KUKA KRL program: MyProgram_137().src

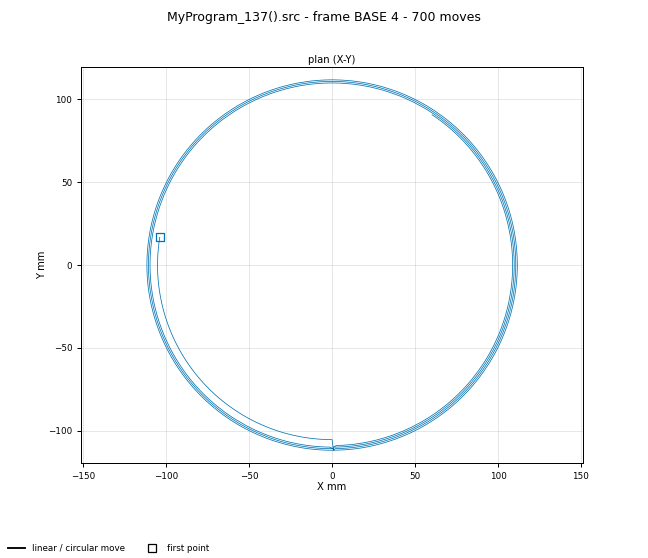
[picture p0: tool path of MyProgram_137().src in frame BASE 4, 700 of 700 moves have a stored position in this frame; points joined in program order, loops and branches not executed]
&ACCESS RVP
&REL 1
&PARAM TEMPLATE = C:\KRC\Roboter\Template\vorgabe
&PARAM EDITMASK = *
DEF MyProgram_137()
; ---- Setting reference (Base) ----
$BASE = BASE_DATA[4]

; --------------------------
; ---- Setting tool (TCP) ----
$TOOL = TOOL_DATA[3]
; --------------------------

$VEL.CP = VEL_APROX_PRINT
Startdeposition()
$VEL.CP = VEL_PRINT
LIN {X -103.9153,Y 16.7331,Z 110,A 166.763,B 24.9342,C -1.8738,E1 24.8417,E2 278.8329} C_DIS
LIN {X -104.4625,Y 12.8836,Z 110,A 168.8977,B 24.9346,C -1.8676,E1 24.8409,E2 276.7001} C_DIS
LIN {X -104.7464,Y 10.3245,Z 110,A 170.3073,B 24.9349,C -1.8633,E1 24.8405,E2 275.2923} C_DIS
LIN {X -104.9675,Y 7.7597,Z 110,A 171.7211,B 24.9352,C -1.8592,E1 24.8401,E2 273.8797} C_DIS
LIN {X -105.1015,Y 5.6308,Z 110,A 172.9515,B 24.9352,C -1.858,E1 24.84,E2 272.6448} C_DIS
LIN {X -105.2376,Y 1.7511,Z 110,A 174.9774,B 24.936,C -1.848,E1 24.8398,E2 270.6305} C_DIS
LIN {X -105.2498,Y -0.7552,Z 110,A 176.4837,B 24.936,C -1.8487,E1 24.8398,E2 269.1135} C_DIS
LIN {X -105.1831,Y -3.8616,Z 110,A 178.2625,B 24.936,C -1.8464,E1 24.84,E2 267.3295} C_DIS
LIN {X -105.0018,Y -7.2556,Z 110,A 179.9647,B 24.9369,C -1.8351,E1 24.8402,E2 265.6439} C_DIS
LIN {X -104.7784,Y -9.9782,Z 110,A -178.5617,B 24.9372,C -1.8299,E1 24.8406,E2 264.1741} C_DIS
LIN {X -104.4634,Y -12.8763,Z 110,A -176.7775,B 24.9371,C -1.8319,E1 24.8412,E2 262.3742} C_DIS
LIN {X -104.0207,Y -16.0526,Z 110,A -175.1402,B 24.9377,C -1.8225,E1 24.8419,E2 260.7497} C_DIS
LIN {X -103.4748,Y -19.271,Z 110,A -173.4007,B 24.9382,C -1.8155,E1 24.8427,E2 259.0165} C_DIS
LIN {X -102.6969,Y -23.0595,Z 110,A -171.2783,B 24.9386,C -1.8096,E1 24.8439,E2 256.8958} C_DIS
LIN {X -102.0023,Y -25.9537,Z 110,A -169.5758,B 24.9388,C -1.8076,E1 24.8451,E2 255.1881} C_DIS
LIN {X -101.2146,Y -28.8725,Z 110,A -167.9294,B 24.9391,C -1.8026,E1 24.8463,E2 253.5441} C_DIS
LIN {X -100.477,Y -31.3431,Z 110,A -166.5162,B 24.9394,C -1.7987,E1 24.8475,E2 252.132} C_DIS
LIN {X -99.3778,Y -34.6711,Z 110,A -164.5611,B 24.9396,C -1.7947,E1 24.8492,E2 250.1753} C_DIS
LIN {X -98.2809,Y -37.67,Z 110,A -162.7314,B 24.9398,C -1.7929,E1 24.851,E2 248.3396} C_DIS
LIN {X -96.9545,Y -40.9612,Z 110,A -160.9726,B 24.9405,C -1.781,E1 24.8529,E2 246.5994} C_DIS
LIN {X -95.6958,Y -43.8259,Z 110,A -159.2509,B 24.9408,C -1.7767,E1 24.8548,E2 244.8784} C_DIS
LIN {X -94.0154,Y -47.3234,Z 110,A -157.1242,B 24.9412,C -1.7713,E1 24.8574,E2 242.7531} C_DIS
LIN {X -92.2133,Y -50.7454,Z 110,A -155.0081,B 24.9416,C -1.7659,E1 24.8602,E2 240.6386} C_DIS
LIN {X -90.2743,Y -54.1198,Z 110,A -152.8768,B 24.9419,C -1.7607,E1 24.8632,E2 238.5087} C_DIS
LIN {X -88.4772,Y -57.0071,Z 110,A -150.9522,B 24.942,C -1.7586,E1 24.8661,E2 236.5793} C_DIS
LIN {X -86.4702,Y -60.0076,Z 110,A -148.9751,B 24.9423,C -1.754,E1 24.8692,E2 234.6033} C_DIS
LIN {X -84.5433,Y -62.6964,Z 110,A -147.1303,B 24.9425,C -1.7512,E1 24.8722,E2 232.7564} C_DIS
LIN {X -82.5713,Y -65.2685,Z 110,A -145.3762,B 24.9428,C -1.7466,E1 24.8752,E2 231.005} C_DIS
LIN {X -80.5409,Y -67.7611,Z 110,A -143.5381,B 24.9428,C -1.7457,E1 24.8785,E2 229.1605} C_DIS
LIN {X -78.4313,Y -70.1892,Z 110,A -141.8851,B 24.9434,C -1.7381,E1 24.8816,E2 227.5181} C_DIS
LIN {X -76.0517,Y -72.7618,Z 110,A -139.8973,B 24.9434,C -1.7369,E1 24.8854,E2 225.5246} C_DIS
LIN {X -73.6749,Y -75.1676,Z 110,A -137.9924,B 24.9436,C -1.7354,E1 24.8892,E2 223.6152} C_DIS
LIN {X -71.1541,Y -77.5569,Z 110,A -136.1922,B 24.944,C -1.7281,E1 24.8928,E2 221.8249} C_DIS
LIN {X -68.4428,Y -79.9602,Z 110,A -134.2214,B 24.9443,C -1.7242,E1 24.897,E2 219.8558} C_DIS
LIN {X -65.975,Y -82.0088,Z 110,A -132.4324,B 24.9443,C -1.7225,E1 24.9008,E2 218.0638} C_DIS
LIN {X -63.2601,Y -84.1199,Z 110,A -130.6012,B 24.9447,C -1.7177,E1 24.9049,E2 216.2377} C_DIS
LIN {X -60.6051,Y -86.0548,Z 110,A -128.8602,B 24.945,C -1.7128,E1 24.9088,E2 214.5022} C_DIS
LIN {X -58.8664,Y -87.2512,Z 110,A -127.6452,B 24.945,C -1.7135,E1 24.9116,E2 213.2815} C_DIS
LIN {X -55.9198,Y -89.1684,Z 110,A -125.7403,B 24.9452,C -1.7102,E1 24.9161,E2 211.3784} C_DIS
LIN {X -53.3923,Y -90.7044,Z 110,A -124.1717,B 24.9454,C -1.7062,E1 24.9199,E2 209.8144} C_DIS
LIN {X -50.7507,Y -92.2105,Z 110,A -122.5116,B 24.9456,C -1.7041,E1 24.9239,E2 208.1545} C_DIS
LIN {X -47.3297,Y -94.0122,Z 110,A -120.4002,B 24.9457,C -1.7016,E1 24.9292,E2 206.0432} C_DIS
LIN {X -44.5872,Y -95.3415,Z 110,A -118.6477,B 24.9457,C -1.7033,E1 24.9336,E2 204.2823} C_DIS
LIN {X -41.4753,Y -96.7378,Z 110,A -116.6757,B 24.9455,C -1.7057,E1 24.9387,E2 202.2999} C_DIS
LIN {X -38.3078,Y -98.0333,Z 110,A -114.9479,B 24.9459,C -1.6986,E1 24.9431,E2 200.585} C_DIS
LIN {X -35.4596,Y -99.1011,Z 110,A -113.3497,B 24.9462,C -1.6949,E1 24.9473,E2 198.9925} C_DIS
LIN {X -32.2801,Y -100.1799,Z 110,A -111.4454,B 24.9461,C -1.6964,E1 24.9524,E2 197.081} C_DIS
LIN {X -29.7694,Y -100.9545,Z 110,A -110.024,B 24.9461,C -1.6951,E1 24.9562,E2 195.6605} C_DIS
LIN {X -26.887,Y -101.7616,Z 110,A -108.4517,B 24.9464,C -1.6918,E1 24.9604,E2 194.0935} C_DIS
LIN {X -23.518,Y -102.5911,Z 110,A -106.5641,B 24.9464,C -1.6908,E1 24.9655,E2 192.2058} C_DIS
LIN {X -20.5482,Y -103.2287,Z 110,A -104.9083,B 24.9464,C -1.6901,E1 24.97,E2 190.5495} C_DIS
LIN {X -18.4552,Y -103.6216,Z 110,A -103.6876,B 24.9464,C -1.6922,E1 24.9734,E2 189.3228} C_DIS
LIN {X -15.4692,Y -104.1109,Z 110,A -101.9398,B 24.9461,C -1.6957,E1 24.9783,E2 187.5651} C_DIS
LIN {X -12.1794,Y -104.545,Z 110,A -100.2029,B 24.9463,C -1.6927,E1 24.983,E2 185.8341} C_DIS
LIN {X -9.4942,Y -104.8231,Z 110,A -98.762,B 24.9463,C -1.6914,E1 24.987,E2 184.3955} C_DIS
LIN {X -6.4614,Y -105.0554,Z 110,A -96.9999,B 24.9461,C -1.6956,E1 24.992,E2 182.6227} C_DIS
LIN {X -3.061,Y -105.2076,Z 110,A -95.3134,B 24.9465,C -1.6892,E1 24.9967,E2 180.9511} C_DIS
LIN {X 0.0042,Y -105.254,Z 110,A -93.6476,B 24.9465,C -1.6894,E1 25.0013,E2 179.2848} C_DIS
LIN {X 0.0042,Y -105.254,Z 110,A -93.6476,B 24.9465,C -1.6894,E1 25.0013,E2 179.2848} C_DIS
Enddeposition()
LIN {X 0.777,Y -111.6543,Z 111,A -93.3875,B 24.9533,C -1.5793,E1 25.0013,E2 179.2857} C_DIS
Startdeposition()
$VEL.CP = VEL_PRINT
LIN {X -3.579,Y -111.5997,Z 111,A -95.9681,B 24.9542,C -1.5643,E1 24.994,E2 181.902} C_DIS
LIN {X -7.9797,Y -111.3724,Z 111,A -98.1296,B 24.9539,C -1.5684,E1 24.988,E2 184.0545} C_DIS
LIN {X -10.4157,Y -111.1702,Z 111,A -99.4838,B 24.9542,C -1.5643,E1 24.9842,E2 185.4191} C_DIS
LIN {X -13.1408,Y -110.8811,Z 111,A -100.8903,B 24.9542,C -1.5645,E1 24.9803,E2 186.8261} C_DIS
LIN {X -17.2131,Y -110.3223,Z 111,A -102.9327,B 24.9539,C -1.5678,E1 24.9747,E2 188.8623} C_DIS
LIN {X -20.4381,Y -109.7727,Z 111,A -104.6115,B 24.9539,C -1.5683,E1 24.9701,E2 190.5416} C_DIS
LIN {X -23.9458,Y -109.0592,Z 111,A -106.4503,B 24.9539,C -1.569,E1 24.965,E2 192.3808} C_DIS
LIN {X -27.1309,Y -108.3128,Z 111,A -108.1308,B 24.9539,C -1.5698,E1 24.9605,E2 194.0617} C_DIS
LIN {X -29.2682,Y -107.7529,Z 111,A -109.3355,B 24.9539,C -1.5676,E1 24.9572,E2 195.2734} C_DIS
LIN {X -32.4129,Y -106.8511,Z 111,A -110.9474,B 24.9537,C -1.5715,E1 24.9529,E2 196.8788} C_DIS
LIN {X -34.5201,Y -106.187,Z 111,A -112.1525,B 24.9538,C -1.5695,E1 24.9497,E2 198.0909} C_DIS
LIN {X -37.1157,Y -105.3078,Z 111,A -113.561,B 24.9538,C -1.5706,E1 24.946,E2 199.4995} C_DIS
LIN {X -40.1856,Y -104.1771,Z 111,A -115.1737,B 24.9535,C -1.5748,E1 24.9418,E2 201.1055} C_DIS
LIN {X -42.7301,Y -103.1596,Z 111,A -116.5831,B 24.9535,C -1.5761,E1 24.9381,E2 202.5151} C_DIS
LIN {X -44.762,Y -102.2921,Z 111,A -117.7889,B 24.9535,C -1.5744,E1 24.935,E2 203.7276} C_DIS
LIN {X -47.385,Y -101.1041,Z 111,A -119.2415,B 24.9534,C -1.5771,E1 24.9313,E2 205.1775} C_DIS
LIN {X -50.2032,Y -99.7366,Z 111,A -120.8124,B 24.9532,C -1.5805,E1 24.9274,E2 206.7442} C_DIS
LIN {X -52.6357,Y -98.4745,Z 111,A -122.2227,B 24.9531,C -1.5822,E1 24.9239,E2 208.1545} C_DIS
LIN {X -55.0366,Y -97.1531,Z 111,A -123.6331,B 24.953,C -1.584,E1 24.9205,E2 209.5648} C_DIS
LIN {X -57.4042,Y -95.7732,Z 111,A -125.0438,B 24.9529,C -1.5859,E1 24.9171,E2 210.9753} C_DIS
LIN {X -59.2869,Y -94.617,Z 111,A -126.2507,B 24.9529,C -1.5847,E1 24.9142,E2 212.1889} C_DIS
LIN {X -62.0345,Y -92.8411,Z 111,A -127.8657,B 24.9526,C -1.5899,E1 24.9105,E2 213.7968} C_DIS
LIN {X -64.2942,Y -91.2908,Z 111,A -129.2769,B 24.9526,C -1.592,E1 24.9072,E2 215.2077} C_DIS
LIN {X -66.0867,Y -89.9992,Z 111,A -130.4845,B 24.9526,C -1.591,E1 24.9045,E2 216.4219} C_DIS
LIN {X -68.4695,Y -88.2007,Z 111,A -131.9236,B 24.9522,C -1.5975,E1 24.9013,E2 217.8508} C_DIS
LIN {X -70.8358,Y -86.3136,Z 111,A -133.5119,B 24.9521,C -1.5989,E1 24.8979,E2 219.4417} C_DIS
LIN {X -73.3327,Y -84.1999,Z 111,A -135.2342,B 24.9521,C -1.6005,E1 24.8942,E2 221.167} C_DIS
LIN {X -75.604,Y -82.1666,Z 111,A -136.7691,B 24.9517,C -1.6048,E1 24.891,E2 222.6978} C_DIS
LIN {X -77.5977,Y -80.2864,Z 111,A -138.1945,B 24.9517,C -1.6069,E1 24.8881,E2 224.1239} C_DIS
LIN {X -79.5446,Y -78.3579,Z 111,A -139.5865,B 24.9514,C -1.6105,E1 24.8854,E2 225.5133} C_DIS
LIN {X -81.8075,Y -75.9953,Z 111,A -141.2811,B 24.9512,C -1.6135,E1 24.8822,E2 227.2081} C_DIS
LIN {X -83.6479,Y -73.9647,Z 111,A -142.6944,B 24.951,C -1.6164,E1 24.8795,E2 228.6208} C_DIS
LIN {X -86.0325,Y -71.1741,Z 111,A -144.5728,B 24.9508,C -1.6211,E1 24.8761,E2 230.4968} C_DIS
LIN {X -88.026,Y -68.6962,Z 111,A -146.2279,B 24.9506,C -1.624,E1 24.8733,E2 232.1526} C_DIS
LIN {X -90.0917,Y -65.9603,Z 111,A -148.0284,B 24.9504,C -1.6268,E1 24.8703,E2 233.9552} C_DIS
LIN {X -91.7698,Y -63.6052,Z 111,A -149.4887,B 24.9501,C -1.6314,E1 24.8679,E2 235.4116} C_DIS
LIN {X -93.3031,Y -61.3339,Z 111,A -150.9028,B 24.9499,C -1.6348,E1 24.8657,E2 236.8248} C_DIS
LIN {X -95.0616,Y -58.5752,Z 111,A -152.5909,B 24.9497,C -1.6388,E1 24.8632,E2 238.512} C_DIS
LIN {X -96.8885,Y -55.497,Z 111,A -154.4387,B 24.9494,C -1.6433,E1 24.8606,E2 240.3585} C_DIS
LIN {X -98.4745,Y -52.6357,Z 111,A -156.3071,B 24.9496,C -1.6405,E1 24.8581,E2 242.2436} C_DIS
LIN {X -100.0741,Y -49.5224,Z 111,A -157.95,B 24.9489,C -1.6515,E1 24.856,E2 243.869} C_DIS
LIN {X -101.2928,Y -46.9796,Z 111,A -159.3903,B 24.9486,C -1.6558,E1 24.8543,E2 245.3067} C_DIS
LIN {X -102.5077,Y -44.2674,Z 111,A -160.8961,B 24.9483,C -1.661,E1 24.8526,E2 246.8087} C_DIS
LIN {X -103.4759,Y -41.9528,Z 111,A -162.2901,B 24.9483,C -1.6606,E1 24.8512,E2 248.2113} C_DIS
LIN {X -104.95,Y -38.1158,Z 111,A -164.4131,B 24.948,C -1.6663,E1 24.8491,E2 250.3326} C_DIS
LIN {X -105.8538,Y -35.5287,Z 111,A -165.8285,B 24.9477,C -1.6702,E1 24.8478,E2 251.7469} C_DIS
LIN {X -107.0898,Y -31.6084,Z 111,A -167.8819,B 24.9472,C -1.6787,E1 24.8461,E2 253.7917} C_DIS
LIN {X -107.9717,Y -28.4581,Z 111,A -169.5719,B 24.9469,C -1.6834,E1 24.8449,E2 255.4804} C_DIS
LIN {X -108.946,Y -24.4646,Z 111,A -171.6954,B 24.9465,C -1.6894,E1 24.8435,E2 257.6021} C_DIS
LIN {X -109.5136,Y -21.7836,Z 111,A -173.1112,B 24.9463,C -1.6934,E1 24.8427,E2 259.0166} C_DIS
LIN {X -110.1536,Y -18.2618,Z 111,A -175.0306,B 24.9461,C -1.6961,E1 24.8418,E2 260.941} C_DIS
LIN {X -110.6433,Y -15.0272,Z 111,A -176.6511,B 24.9456,C -1.7036,E1 24.8411,E2 262.5532} C_DIS
LIN {X -110.9788,Y -12.3073,Z 111,A -178.0669,B 24.9453,C -1.7077,E1 24.8407,E2 263.9677} C_DIS
LIN {X -111.3566,Y -8.2142,Z 111,A 179.8089,B 24.9449,C -1.7139,E1 24.8402,E2 266.0899} C_DIS
LIN {X -111.5246,Y -5.4789,Z 111,A 178.3928,B 24.9447,C -1.7181,E1 24.8399,E2 267.5046} C_DIS
LIN {X -111.6255,Y -2.7403,Z 111,A 176.9767,B 24.9444,C -1.7222,E1 24.8399,E2 268.9194} C_DIS
LIN {X -111.6594,Y 0.1303,Z 111,A 175.3018,B 24.9446,C -1.7193,E1 24.8398,E2 270.6114} C_DIS
LIN {X -111.5997,Y 3.579,Z 111,A 173.6409,B 24.944,C -1.7292,E1 24.8399,E2 272.2585} C_DIS
LIN {X -111.4783,Y 6.3167,Z 111,A 172.2247,B 24.9437,C -1.7334,E1 24.8401,E2 273.6732} C_DIS
LIN {X -111.1702,Y 10.4157,Z 111,A 170.1004,B 24.9433,C -1.7397,E1 24.8406,E2 275.7954} C_DIS
LIN {X -110.8811,Y 13.1408,Z 111,A 168.6843,B 24.943,C -1.7439,E1 24.841,E2 277.2099} C_DIS
LIN {X -110.3223,Y 17.2131,Z 111,A 166.56,B 24.9426,C -1.7501,E1 24.8419,E2 279.332} C_DIS
LIN {X -109.8667,Y 19.9154,Z 111,A 165.144,B 24.9423,C -1.7543,E1 24.8426,E2 280.7465} C_DIS
LIN {X -109.0592,Y 23.9458,Z 111,A 163.0198,B 24.9419,C -1.7605,E1 24.8438,E2 282.8684} C_DIS
LIN {X -108.4387,Y 26.615,Z 111,A 161.604,B 24.9416,C -1.7646,E1 24.8447,E2 284.2827} C_DIS
LIN {X -107.7529,Y 29.2682,Z 111,A 160.1878,B 24.9414,C -1.7687,E1 24.8457,E2 285.6974} C_DIS
LIN {X -107.0021,Y 31.9038,Z 111,A 158.7719,B 24.9411,C -1.7728,E1 24.8468,E2 287.1117} C_DIS
LIN {X -106.0235,Y 35.0254,Z 111,A 157.1514,B 24.9406,C -1.7803,E1 24.8482,E2 288.7237} C_DIS
LIN {X -104.8444,Y 38.4052,Z 111,A 155.3114,B 24.9402,C -1.7859,E1 24.8499,E2 290.5607} C_DIS
LIN {X -103.8703,Y 40.9666,Z 111,A 153.8864,B 24.94,C -1.7895,E1 24.8514,E2 291.985} C_DIS
LIN {X -102.8337,Y 43.5034,Z 111,A 152.4012,B 24.9399,C -1.7908,E1 24.853,E2 293.4754} C_DIS
LIN {X -101.5169,Y 46.4981,Z 111,A 150.7811,B 24.9394,C -1.7981,E1 24.8548,E2 295.0869} C_DIS
LIN {X -100.5546,Y 48.5396,Z 111,A 149.5559,B 24.9394,C -1.7991,E1 24.8563,E2 296.3165} C_DIS
LIN {X -99.3547,Y 50.9504,Z 111,A 148.1547,B 24.9391,C -1.8025,E1 24.858,E2 297.7172} C_DIS
LIN {X -97.8212,Y 53.8402,Z 111,A 146.5354,B 24.9386,C -1.8097,E1 24.8602,E2 299.328} C_DIS
LIN {X -96.4704,Y 56.2246,Z 111,A 145.1199,B 24.9384,C -1.8134,E1 24.8621,E2 300.7419} C_DIS
LIN {X -94.617,Y 59.2869,Z 111,A 143.2716,B 24.938,C -1.8182,E1 24.8648,E2 302.5881} C_DIS
LIN {X -92.8411,Y 62.0345,Z 111,A 141.5826,B 24.9377,C -1.8225,E1 24.8674,E2 304.2753} C_DIS
LIN {X -91.3255,Y 64.2443,Z 111,A 140.198,B 24.9375,C -1.826,E1 24.8696,E2 305.6585} C_DIS
LIN {X -89.6854,Y 66.5152,Z 111,A 138.7532,B 24.9373,C -1.8296,E1 24.872,E2 307.1017} C_DIS
LIN {X -87.1764,Y 69.7712,Z 111,A 136.6316,B 24.9369,C -1.8348,E1 24.8756,E2 309.221} C_DIS
LIN {X -84.5998,Y 72.8734,Z 111,A 134.5688,B 24.9365,C -1.8405,E1 24.8793,E2 311.2798} C_DIS
LIN {X -82.1666,Y 75.604,Z 111,A 132.6633,B 24.9363,C -1.8441,E1 24.8829,E2 313.185} C_DIS
LIN {X -80.2864,Y 77.5977,Z 111,A 131.1797,B 24.9363,C -1.8446,E1 24.8858,E2 314.6739} C_DIS
LIN {X -78.3579,Y 79.5446,Z 111,A 129.7661,B 24.936,C -1.8477,E1 24.8886,E2 316.086} C_DIS
LIN {X -75.9953,Y 81.8075,Z 111,A 128.1485,B 24.9356,C -1.8541,E1 24.8918,E2 317.6953} C_DIS
LIN {X -73.9647,Y 83.6479,Z 111,A 126.735,B 24.9354,C -1.857,E1 24.8948,E2 319.1073} C_DIS
LIN {X -71.8896,Y 85.4379,Z 111,A 125.3222,B 24.9352,C -1.8599,E1 24.8978,E2 320.5187} C_DIS
LIN {X -68.6962,Y 88.026,Z 111,A 123.2028,B 24.9349,C -1.8641,E1 24.9024,E2 322.636} C_DIS
LIN {X -65.4097,Y 90.4949,Z 111,A 121.0837,B 24.9346,C -1.8681,E1 24.9071,E2 324.7531} C_DIS
LIN {X -62.4742,Y 92.5434,Z 111,A 119.2389,B 24.9343,C -1.8716,E1 24.9114,E2 326.596} C_DIS
LIN {X -59.7374,Y 94.3356,Z 111,A 117.3931,B 24.9346,C -1.8682,E1 24.9157,E2 328.4558} C_DIS
LIN {X -56.7789,Y 96.1428,Z 111,A 115.7441,B 24.934,C -1.8766,E1 24.9196,E2 330.0899} C_DIS
LIN {X -53.8726,Y 97.8031,Z 111,A 114.0527,B 24.9337,C -1.8806,E1 24.9237,E2 331.7766} C_DIS
LIN {X -50.7454,Y 99.4595,Z 111,A 112.2048,B 24.9336,C -1.8824,E1 24.9283,E2 333.6253} C_DIS
LIN {X -48.2191,Y 100.7086,Z 111,A 110.7692,B 24.9334,C -1.8851,E1 24.9319,E2 335.0581} C_DIS
LIN {X -45.7331,Y 101.8616,Z 111,A 109.2886,B 24.9334,C -1.8843,E1 24.9357,E2 336.5443} C_DIS
LIN {X -42.7301,Y 103.1596,Z 111,A 107.6743,B 24.9331,C -1.8893,E1 24.9398,E2 338.1506} C_DIS
LIN {X -40.1856,Y 104.1771,Z 111,A 106.264,B 24.933,C -1.891,E1 24.9435,E2 339.5598} C_DIS
LIN {X -36.3239,Y 105.5857,Z 111,A 103.9696,B 24.9333,C -1.8863,E1 24.9496,E2 341.87} C_DIS
LIN {X -33.0876,Y 106.6419,Z 111,A 102.3597,B 24.9328,C -1.8939,E1 24.9538,E2 343.4647} C_DIS
LIN {X -30.2919,Y 107.4696,Z 111,A 100.828,B 24.9328,C -1.8941,E1 24.9579,E2 344.9984} C_DIS
LIN {X -26.3157,Y 108.5117,Z 111,A 98.7142,B 24.9326,C -1.896,E1 24.9636,E2 347.1108} C_DIS
LIN {X -23.1259,Y 109.238,Z 111,A 97.1015,B 24.9323,C -1.9001,E1 24.968,E2 348.7157} C_DIS
LIN {X -20.4381,Y 109.7727,Z 111,A 95.6931,B 24.9323,C -1.9011,E1 24.9719,E2 350.1232} C_DIS
LIN {X -16.3838,Y 110.4506,Z 111,A 93.5804,B 24.9321,C -1.9025,E1 24.9777,E2 352.2345} C_DIS
LIN {X -14.195,Y 110.7511,Z 111,A 92.3757,B 24.9323,C -1.9003,E1 24.981,E2 353.4453} C_DIS
LIN {X -11.4727,Y 111.0661,Z 111,A 90.9678,B 24.9323,C -1.901,E1 24.985,E2 354.8524} C_DIS
LIN {X -7.9091,Y 111.3772,Z 111,A 89.1149,B 24.9323,C -1.9011,E1 24.9901,E2 356.7059} C_DIS
LIN {X -4.6405,Y 111.5606,Z 111,A 87.4491,B 24.9322,C -1.9023,E1 24.9948,E2 358.3693} C_DIS
LIN {X -1.3702,Y 111.6507,Z 111,A 85.839,B 24.9319,C -1.9056,E1 24.9992,E2 359.9719} C_DIS
LIN {X 1.3702,Y 111.6507,Z 111,A 84.432,B 24.9319,C -1.9058,E1 25.0032,E2 361.3783} C_DIS
LIN {X 5.4789,Y 111.5246,Z 111,A 82.3223,B 24.9319,C -1.9059,E1 25.009,E2 363.487} C_DIS
LIN {X 9.0506,Y 111.2897,Z 111,A 80.4855,B 24.9319,C -1.9059,E1 25.0142,E2 365.323} C_DIS
LIN {X 12.3073,Y 110.9788,Z 111,A 78.8073,B 24.9319,C -1.9056,E1 25.0188,E2 367.0007} C_DIS
LIN {X 15.0272,Y 110.6433,Z 111,A 77.402,B 24.9319,C -1.9054,E1 25.0227,E2 368.4056} C_DIS
LIN {X 19.0895,Y 110.0152,Z 111,A 75.2938,B 24.9319,C -1.9047,E1 25.0285,E2 370.5132} C_DIS
LIN {X 21.7836,Y 109.5136,Z 111,A 73.7103,B 24.9326,C -1.8967,E1 25.0329,E2 372.1138} C_DIS
LIN {X 25.1144,Y 108.7959,Z 111,A 72.1055,B 24.9322,C -1.9019,E1 25.0372,E2 373.7042} C_DIS
LIN {X 27.9437,Y 108.1039,Z 111,A 70.6494,B 24.9322,C -1.9026,E1 25.0412,E2 375.1564} C_DIS
LIN {X 31.0993,Y 107.2408,Z 111,A 68.9737,B 24.9322,C -1.9016,E1 25.0457,E2 376.8319} C_DIS
LIN {X 33.6847,Y 106.4568,Z 111,A 67.5886,B 24.9322,C -1.9005,E1 25.0494,E2 378.2168} C_DIS
LIN {X 36.165,Y 105.6392,Z 111,A 66.243,B 24.9324,C -1.8992,E1 25.0529,E2 379.563} C_DIS
LIN {X 38.9041,Y 104.6624,Z 111,A 64.7622,B 24.9324,C -1.8983,E1 25.0568,E2 381.0429} C_DIS
LIN {X 42.2382,Y 103.3598,Z 111,A 62.9293,B 24.9326,C -1.8966,E1 25.0616,E2 382.8756} C_DIS
LIN {X 45.2489,Y 102.0798,Z 111,A 61.2547,B 24.9326,C -1.8949,E1 25.0659,E2 384.5503} C_DIS
LIN {X 47.67,Y 100.9714,Z 111,A 59.8899,B 24.9328,C -1.8934,E1 25.0693,E2 385.9153} C_DIS
LIN {X 50.0896,Y 99.7929,Z 111,A 58.5265,B 24.9328,C -1.8924,E1 25.0727,E2 387.2774} C_DIS
LIN {X 52.1658,Y 98.722,Z 111,A 57.2499,B 24.9332,C -1.8875,E1 25.0759,E2 388.5619} C_DIS
LIN {X 54.5729,Y 97.4121,Z 111,A 55.8479,B 24.9333,C -1.8857,E1 25.0793,E2 389.9641} C_DIS
LIN {X 57.4042,Y 95.7732,Z 111,A 54.2437,B 24.9333,C -1.8864,E1 25.0832,E2 391.5618} C_DIS
LIN {X 59.7374,Y 94.3356,Z 111,A 52.8421,B 24.9334,C -1.8844,E1 25.0865,E2 392.9636} C_DIS
LIN {X 62.0345,Y 92.8411,Z 111,A 51.4407,B 24.9336,C -1.8823,E1 25.0898,E2 394.3652} C_DIS
LIN {X 64.2942,Y 91.2908,Z 111,A 50.0397,B 24.9337,C -1.8802,E1 25.093,E2 395.7665} C_DIS
LIN {X 66.0867,Y 89.9992,Z 111,A 48.841,B 24.9341,C -1.8754,E1 25.0957,E2 396.9722} C_DIS
LIN {X 68.2755,Y 88.3502,Z 111,A 47.4405,B 24.9342,C -1.8731,E1 25.0988,E2 398.3731} C_DIS
LIN {X 71.2442,Y 85.9742,Z 111,A 45.5515,B 24.9342,C -1.8722,E1 25.1029,E2 400.2571} C_DIS
LIN {X 73.5647,Y 83.9972,Z 111,A 43.9393,B 24.9347,C -1.867,E1 25.1063,E2 401.8752} C_DIS
LIN {X 75.9953,Y 81.8075,Z 111,A 42.1588,B 24.9352,C -1.8591,E1 25.11,E2 403.6672} C_DIS
LIN {X 78.4907,Y 79.4134,Z 111,A 40.5456,B 24.935,C -1.8624,E1 25.1132,E2 405.2658} C_DIS
LIN {X 80.8688,Y 76.9935,Z 111,A 38.8376,B 24.9351,C -1.86,E1 25.1165,E2 406.9722} C_DIS
LIN {X 82.7339,Y 74.9857,Z 111,A 37.4382,B 24.9353,C -1.8572,E1 25.1192,E2 408.3722} C_DIS
LIN {X 85.0935,Y 72.2939,Z 111,A 35.5413,B 24.9358,C -1.8503,E1 25.1227,E2 410.2767} C_DIS
LIN {X 87.6967,Y 69.1129,Z 111,A 33.5116,B 24.9359,C -1.8488,E1 25.1262,E2 412.3006} C_DIS
LIN {X 89.4688,Y 66.8036,Z 111,A 32.0496,B 24.9361,C -1.8465,E1 25.1287,E2 413.761} C_DIS
LIN {X 91.2908,Y 64.2942,Z 111,A 30.4433,B 24.9364,C -1.8418,E1 25.1313,E2 415.3706} C_DIS
LIN {X 92.8411,Y 62.0345,Z 111,A 29.0448,B 24.9366,C -1.8385,E1 25.1335,E2 416.7699} C_DIS
LIN {X 94.7802,Y 59.0256,Z 111,A 27.2182,B 24.9369,C -1.8342,E1 25.1362,E2 418.5975} C_DIS
LIN {X 96.2002,Y 56.6818,Z 111,A 25.8201,B 24.9372,C -1.8308,E1 25.1382,E2 419.9966} C_DIS
LIN {X 97.8212,Y 53.8402,Z 111,A 24.151,B 24.9375,C -1.8266,E1 25.1405,E2 421.6668} C_DIS
LIN {X 99.4949,Y 50.6761,Z 111,A 22.261,B 24.938,C -1.8191,E1 25.143,E2 423.5644} C_DIS
LIN {X 101.1628,Y 47.2589,Z 111,A 20.34,B 24.9383,C -1.8149,E1 25.1453,E2 425.485} C_DIS
LIN {X 102.4152,Y 44.4796,Z 111,A 18.8311,B 24.9383,C -1.8129,E1 25.147,E2 426.9904} C_DIS
LIN {X 103.4759,Y 41.9528,Z 111,A 17.3649,B 24.9389,C -1.8061,E1 25.1486,E2 428.4646} C_DIS
LIN {X 104.95,Y 38.1158,Z 111,A 15.2688,B 24.9392,C -1.8005,E1 25.1506,E2 430.5623} C_DIS
LIN {X 105.8538,Y 35.5287,Z 111,A 13.8716,B 24.9395,C -1.7966,E1 25.1519,E2 431.9607} C_DIS
LIN {X 106.6938,Y 32.9202,Z 111,A 12.4744,B 24.9398,C -1.7928,E1 25.153,E2 433.359} C_DIS
LIN {X 107.4696,Y 30.2919,Z 111,A 11.0775,B 24.94,C -1.7889,E1 25.1541,E2 434.7571} C_DIS
LIN {X 108.5117,Y 26.3157,Z 111,A 8.9821,B 24.9404,C -1.783,E1 25.1556,E2 436.8543} C_DIS
LIN {X 109.238,Y 23.1259,Z 111,A 7.3833,B 24.9405,C -1.7813,E1 25.1565,E2 438.4478} C_DIS
LIN {X 109.9949,Y 19.2024,Z 111,A 5.3703,B 24.9408,C -1.7766,E1 25.1576,E2 440.4602} C_DIS
LIN {X 110.4506,Y 16.3838,Z 111,A 3.8917,B 24.9412,C -1.7713,E1 25.1582,E2 441.9426} C_DIS
LIN {X 110.7511,Y 14.195,Z 111,A 2.6969,B 24.9416,C -1.7649,E1 25.1586,E2 443.1453} C_DIS
LIN {X 111.231,Y 9.7569,Z 111,A 0.4812,B 24.9419,C -1.761,E1 25.1593,E2 445.3572} C_DIS
LIN {X 111.4131,Y 7.3769,Z 111,A -0.7946,B 24.9423,C -1.7547,E1 25.1595,E2 446.6401} C_DIS
LIN {X 111.5606,Y 4.6405,Z 111,A -2.1911,B 24.9426,C -1.7506,E1 25.1597,E2 448.038} C_DIS
LIN {X 111.6507,Y 1.3702,Z 111,A -3.7448,B 24.9426,C -1.7508,E1 25.1597,E2 449.582} C_DIS
LIN {X 111.6507,Y -1.3702,Z 111,A -5.1859,B 24.943,C -1.7446,E1 25.1597,E2 451.0291} C_DIS
LIN {X 111.5372,Y -5.1852,Z 111,A -7.1023,B 24.9432,C -1.7402,E1 25.1596,E2 452.9446} C_DIS
LIN {X 111.3566,Y -8.2142,Z 111,A -8.677,B 24.9436,C -1.7343,E1 25.1593,E2 454.5237} C_DIS
LIN {X 110.9788,Y -12.3073,Z 111,A -10.7716,B 24.944,C -1.7281,E1 25.1587,E2 456.6206} C_DIS
LIN {X 110.6433,Y -15.0272,Z 111,A -12.1679,B 24.9443,C -1.724,E1 25.1582,E2 458.0183} C_DIS
LIN {X 110.0152,Y -19.0894,Z 111,A -14.2629,B 24.9447,C -1.7178,E1 25.1573,E2 460.1156} C_DIS
LIN {X 109.3448,Y -22.6056,Z 111,A -16.087,B 24.945,C -1.7125,E1 25.1563,E2 461.9416} C_DIS
LIN {X 108.7571,Y -25.2823,Z 111,A -17.5523,B 24.9455,C -1.7053,E1 25.1554,E2 463.4154} C_DIS
LIN {X 107.9717,Y -28.4581,Z 111,A -19.1508,B 24.9456,C -1.7035,E1 25.1543,E2 465.0089} C_DIS
LIN {X 107.2408,Y -31.0993,Z 111,A -20.5472,B 24.9459,C -1.6995,E1 25.1532,E2 466.4068} C_DIS
LIN {X 106.478,Y -33.6163,Z 111,A -21.8652,B 24.9461,C -1.6967,E1 25.1521,E2 467.7239} C_DIS
LIN {X 105.5857,Y -36.3239,Z 111,A -23.3408,B 24.9464,C -1.6915,E1 25.1508,E2 469.2034} C_DIS
LIN {X 104.6624,Y -38.9041,Z 111,A -24.7379,B 24.9466,C -1.6875,E1 25.1495,E2 470.6021} C_DIS
LIN {X 103.8703,Y -40.9666,Z 111,A -25.9328,B 24.947,C -1.6812,E1 25.1483,E2 471.8052} C_DIS
LIN {X 102.6274,Y -43.9928,Z 111,A -27.5315,B 24.9471,C -1.6796,E1 25.1466,E2 473.3988} C_DIS
LIN {X 101.0006,Y -47.6073,Z 111,A -29.5589,B 24.9475,C -1.6737,E1 25.1442,E2 475.4292} C_DIS
LIN {X 99.7366,Y -50.2032,Z 111,A -31.0244,B 24.9477,C -1.67,E1 25.1424,E2 476.8956} C_DIS
LIN {X 98.4745,Y -52.6357,Z 111,A -32.4219,B 24.948,C -1.6662,E1 25.1406,E2 478.2947} C_DIS
LIN {X 97.1531,Y -55.0366,Z 111,A -33.8191,B 24.9482,C -1.6625,E1 25.1387,E2 479.6934} C_DIS
LIN {X 95.7732,Y -57.4042,Z 111,A -35.2166,B 24.9484,C -1.6588,E1 25.1367,E2 481.0925} C_DIS
LIN {X 94.617,Y -59.2869,Z 111,A -36.4122,B 24.9488,C -1.6528,E1 25.1349,E2 482.2961} C_DIS
LIN {X 92.8411,Y -62.0345,Z 111,A -38.0118,B 24.9488,C -1.6515,E1 25.1325,E2 483.8908} C_DIS
LIN {X 91.5069,Y -63.9834,Z 111,A -39.2547,B 24.9492,C -1.6468,E1 25.1305,E2 485.1387} C_DIS
LIN {X 88.9342,Y -67.5152,Z 111,A -41.4502,B 24.9494,C -1.6427,E1 25.1268,E2 487.3333} C_DIS
LIN {X 87.5057,Y -69.3546,Z 111,A -42.7029,B 24.9498,C -1.6369,E1 25.1247,E2 488.5937} C_DIS
LIN {X 84.9016,Y -72.5191,Z 111,A -44.7967,B 24.9501,C -1.6318,E1 25.1209,E2 490.6901} C_DIS
LIN {X 82.1666,Y -75.604,Z 111,A -46.8291,B 24.9502,C -1.6301,E1 25.1171,E2 492.7174} C_DIS
LIN {X 80.2864,Y -77.5977,Z 111,A -48.2967,B 24.9506,C -1.6238,E1 25.1143,E2 494.1935} C_DIS
LIN {X 77.1015,Y -80.7646,Z 111,A -50.5276,B 24.9507,C -1.6215,E1 25.1098,E2 496.4206} C_DIS
LIN {X 74.9857,Y -82.7339,Z 111,A -51.9962,B 24.9509,C -1.6186,E1 25.1068,E2 497.89} C_DIS
LIN {X 72.2939,Y -85.0935,Z 111,A -53.8932,B 24.9513,C -1.6117,E1 25.1028,E2 499.7957} C_DIS
LIN {X 70.1838,Y -86.842,Z 111,A -55.2926,B 24.9515,C -1.6089,E1 25.0998,E2 501.1966} C_DIS
LIN {X 66.9399,Y -89.3664,Z 111,A -57.392,B 24.9517,C -1.6048,E1 25.0951,E2 503.298} C_DIS
LIN {X 63.6052,Y -91.7698,Z 111,A -59.4233,B 24.9518,C -1.6038,E1 25.0905,E2 505.3244} C_DIS
LIN {X 61.3339,Y -93.3031,Z 111,A -60.8235,B 24.952,C -1.6013,E1 25.0872,E2 506.7259} C_DIS
LIN {X 58.5752,Y -95.0616,Z 111,A -62.4952,B 24.9521,C -1.5984,E1 25.0833,E2 508.3992} C_DIS
LIN {X 55.497,Y -96.8885,Z 111,A -64.325,B 24.9523,C -1.5953,E1 25.0789,E2 510.2306} C_DIS
LIN {X 53.1026,Y -98.2213,Z 111,A -65.7258,B 24.9524,C -1.5931,E1 25.0754,E2 511.6326} C_DIS
LIN {X 50.2032,Y -99.7366,Z 111,A -67.3985,B 24.9526,C -1.5905,E1 25.0713,E2 513.3069} C_DIS
LIN {X 47.1297,Y -101.2229,Z 111,A -69.1793,B 24.9528,C -1.5864,E1 25.0668,E2 515.0926} C_DIS
LIN {X 44.6548,Y -102.3388,Z 111,A -70.574,B 24.953,C -1.5842,E1 25.0632,E2 516.4891} C_DIS
LIN {X 41.9528,Y -103.4759,Z 111,A -72.1015,B 24.9532,C -1.581,E1 25.0593,E2 518.0206} C_DIS
LIN {X 38.1158,Y -104.95,Z 111,A -74.2048,B 24.9533,C -1.5784,E1 25.0538,E2 520.1256} C_DIS
LIN {X 34.5201,Y -106.187,Z 111,A -76.129,B 24.9533,C -1.5771,E1 25.0487,E2 522.0492} C_DIS
LIN {X 31.6084,Y -107.0898,Z 111,A -77.6421,B 24.9533,C -1.5775,E1 25.0446,E2 523.5585} C_DIS
LIN {X 28.4581,Y -107.9717,Z 111,A -79.317,B 24.9535,C -1.5759,E1 25.0401,E2 525.2347} C_DIS
LIN {X 24.4646,Y -108.946,Z 111,A -81.4218,B 24.9535,C -1.574,E1 25.0344,E2 527.341} C_DIS
LIN {X 21.7836,Y -109.5136,Z 111,A -82.8254,B 24.9536,C -1.5729,E1 25.0306,E2 528.7456} C_DIS
LIN {X 18.2618,Y -110.1536,Z 111,A -84.6812,B 24.9538,C -1.5706,E1 25.0254,E2 530.6047} C_DIS
LIN {X 15.0272,Y -110.6433,Z 111,A -86.3355,B 24.9538,C -1.5705,E1 25.0209,E2 532.2577} C_DIS
LIN {X 12.3073,Y -110.9788,Z 111,A -87.7396,B 24.9538,C -1.5697,E1 25.017,E2 533.6627} C_DIS
LIN {X 9.5801,Y -111.2474,Z 111,A -89.1445,B 24.9538,C -1.569,E1 25.0131,E2 535.0683} C_DIS
LIN {X 7.3769,Y -111.4131,Z 111,A -90.3463,B 24.9541,C -1.5656,E1 25.0097,E2 536.2776} C_DIS
LIN {X 2.9709,Y -111.6184,Z 111,A -92.5543,B 24.954,C -1.5672,E1 25.0035,E2 538.4815} C_DIS
LIN {X 0.777,Y -111.6543,Z 111,A -93.3874,B 24.9533,C -1.5793,E1 25.0013,E2 539.2857} C_DIS
Enddeposition()
LIN {X 0.777,Y -111.6543,Z 111,A -93.3874,B 24.9533,C -1.5793,E1 25.0013,E2 539.2857} C_DIS
Startdeposition()
$VEL.CP = VEL_PRINT
LIN {X 1.8427,Y -110.7045,Z 111,A -92.4705,B 24.9513,C -1.6113,E1 25.0041,E2 538.2929} C_DIS
LIN {X 4.7468,Y -110.6179,Z 111,A -90.9452,B 24.9513,C -1.6128,E1 25.0083,E2 536.7645} C_DIS
LIN {X 8.4678,Y -110.396,Z 111,A -89.0293,B 24.9513,C -1.6131,E1 25.0137,E2 534.8488} C_DIS
LIN {X 11.6041,Y -110.1099,Z 111,A -87.3617,B 24.9511,C -1.6156,E1 25.0183,E2 533.1763} C_DIS
LIN {X 15.8276,Y -109.5828,Z 111,A -85.0766,B 24.9508,C -1.6206,E1 25.0247,E2 530.8812} C_DIS
LIN {X 19.7657,Y -108.9412,Z 111,A -83.0131,B 24.9507,C -1.6222,E1 25.0304,E2 528.8162} C_DIS
LIN {X 23.5821,Y -108.1792,Z 111,A -81.1085,B 24.9509,C -1.6193,E1 25.0355,E2 526.921} C_DIS
LIN {X 28.3833,Y -107.021,Z 111,A -77.9347,B 24.9491,C -1.6488,E1 25.0443,E2 523.682} C_DIS
LIN {X 32.492,Y -105.8452,Z 111,A -76.4905,B 24.951,C -1.6178,E1 25.048,E2 522.3136} C_DIS
LIN {X 36.6026,Y -104.4945,Z 111,A -74.1107,B 24.9504,C -1.6268,E1 25.0543,E2 519.9174} C_DIS
LIN {X 40.2287,Y -103.1531,Z 111,A -72.095,B 24.9502,C -1.6301,E1 25.0596,E2 517.898} C_DIS
LIN {X 43.5309,Y -101.8049,Z 111,A -70.0324,B 24.9495,C -1.6424,E1 25.0649,E2 515.8113} C_DIS
LIN {X 47.8262,Y -99.8575,Z 111,A -66.4931,B 24.9461,C -1.6953,E1 25.0742,E2 512.1561} C_DIS
LIN {X 54.4727,Y -96.3944,Z 111,A -64.1089,B 24.9499,C -1.6354,E1 25.0796,E2 509.9205} C_DIS
LIN {X 57.3577,Y -94.7046,Z 111,A -62.271,B 24.9494,C -1.6434,E1 25.0841,E2 508.0694} C_DIS
LIN {X 60.3386,Y -92.8358,Z 111,A -60.3736,B 24.949,C -1.6503,E1 25.0886,E2 506.1618} C_DIS
LIN {X 63.1611,Y -90.9369,Z 111,A -58.7657,B 24.9492,C -1.6471,E1 25.0922,E2 504.5669} C_DIS
LIN {X 65.86,Y -89.0034,Z 111,A -57.0766,B 24.949,C -1.6494,E1 25.096,E2 502.8783} C_DIS
LIN {X 67.8704,Y -87.479,Z 111,A -55.6858,B 24.9486,C -1.656,E1 25.0991,E2 501.4769} C_DIS
LIN {X 70.4578,Y -85.409,Z 111,A -53.9321,B 24.9483,C -1.6616,E1 25.103,E2 499.7168} C_DIS
LIN {X 72.9557,Y -83.2847,Z 111,A -52.3071,B 24.9483,C -1.6623,E1 25.1064,E2 498.0965} C_DIS
LIN {X 76.3471,Y -80.1896,Z 111,A -50.0077,B 24.9481,C -1.6644,E1 25.1111,E2 495.8013} C_DIS
LIN {X 78.6771,Y -77.9024,Z 111,A -48.2269,B 24.9476,C -1.6727,E1 25.1146,E2 494.0086} C_DIS
LIN {X 80.9534,Y -75.5353,Z 111,A -46.4192,B 24.947,C -1.6818,E1 25.1181,E2 492.1872} C_DIS
LIN {X 83.5629,Y -72.6371,Z 111,A -44.4882,B 24.947,C -1.6831,E1 25.1217,E2 490.2618} C_DIS
LIN {X 86.2598,Y -69.4136,Z 111,A -42.295,B 24.9465,C -1.6897,E1 25.1256,E2 488.0632} C_DIS
LIN {X 88.4652,Y -66.579,Z 111,A -40.536,B 24.9465,C -1.6903,E1 25.1285,E2 486.3112} C_DIS
LIN {X 90.6999,Y -63.502,Z 111,A -38.39,B 24.9456,C -1.7038,E1 25.1321,E2 484.1437} C_DIS
LIN {X 93.5439,Y -59.2355,Z 111,A -35.5138,B 24.9445,C -1.7214,E1 25.1365,E2 481.2403} C_DIS
LIN {X 95.2986,Y -56.3651,Z 111,A -34.1396,B 24.9452,C -1.7099,E1 25.1384,E2 479.9005} C_DIS
LIN {X 96.8387,Y -53.677,Z 111,A -32.6098,B 24.9452,C -1.7112,E1 25.1405,E2 478.3754} C_DIS
LIN {X 98.5706,Y -50.425,Z 111,A -30.7078,B 24.9448,C -1.7167,E1 25.1429,E2 476.4705} C_DIS
LIN {X 100.0463,Y -47.4333,Z 111,A -28.89,B 24.9442,C -1.7261,E1 25.1451,E2 474.6404} C_DIS
LIN {X 101.5342,Y -44.155,Z 111,A -27.1696,B 24.9442,C -1.7253,E1 25.1471,E2 472.9312} C_DIS
LIN {X 102.93,Y -40.7966,Z 111,A -25.2913,B 24.9438,C -1.7309,E1 25.149,E2 471.05} C_DIS
LIN {X 105.0266,Y -35.0481,Z 111,A -22.0485,B 24.943,C -1.7443,E1 25.1521,E2 467.7939} C_DIS
LIN {X 106.3328,Y -30.8644,Z 111,A -19.8234,B 24.9426,C -1.7495,E1 25.1539,E2 465.5692} C_DIS
LIN {X 107.1889,Y -27.7383,Z 111,A -18.2173,B 24.9425,C -1.7517,E1 25.155,E2 463.9672} C_DIS
LIN {X 107.9293,Y -24.7013,Z 111,A -16.5412,B 24.942,C -1.7595,E1 25.1561,E2 462.2823} C_DIS
LIN {X 108.6993,Y -21.055,Z 111,A -14.7011,B 24.9418,C -1.7617,E1 25.1571,E2 460.4478} C_DIS
LIN {X 109.4054,Y -17.0093,Z 111,A -12.5847,B 24.9414,C -1.7682,E1 25.1581,E2 458.3286} C_DIS
LIN {X 109.9148,Y -13.3338,Z 111,A -10.6273,B 24.9409,C -1.7761,E1 25.1588,E2 456.3641} C_DIS
LIN {X 110.3146,Y -9.4855,Z 111,A -8.5689,B 24.9403,C -1.7852,E1 25.1593,E2 454.2964} C_DIS
LIN {X 110.5911,Y -5.3696,Z 111,A -6.4641,B 24.9399,C -1.7907,E1 25.1597,E2 452.1911} C_DIS
LIN {X 110.709,Y -1.6001,Z 111,A -4.6273,B 24.9399,C -1.7919,E1 25.1597,E2 450.3625} C_DIS
LIN {X 110.7002,Y 2.0748,Z 111,A -2.6825,B 24.9393,C -1.8,E1 25.1597,E2 448.4101} C_DIS
LIN {X 110.5587,Y 5.9701,Z 111,A -0.7555,B 24.9391,C -1.8024,E1 25.1595,E2 446.4888} C_DIS
LIN {X 110.3084,Y 9.5547,Z 111,A 1.2185,B 24.9383,C -1.8136,E1 25.159,E2 444.5003} C_DIS
LIN {X 109.9518,Y 13.0177,Z 111,A 2.8634,B 24.9384,C -1.8123,E1 25.1585,E2 442.8681} C_DIS
LIN {X 109.4819,Y 16.5145,Z 111,A 4.7394,B 24.9379,C -1.8203,E1 25.1578,E2 440.9842} C_DIS
LIN {X 108.9805,Y 19.5474,Z 111,A 6.3471,B 24.9375,C -1.8262,E1 25.157,E2 439.3722} C_DIS
LIN {X 108.1929,Y 23.5192,Z 111,A 8.3913,B 24.9372,C -1.8304,E1 25.1559,E2 437.3299} C_DIS
LIN {X 107.5558,Y 26.2793,Z 111,A 9.933,B 24.9366,C -1.8384,E1 25.1549,E2 435.7782} C_DIS
LIN {X 106.2089,Y 31.282,Z 111,A 12.8346,B 24.9354,C -1.8566,E1 25.1526,E2 432.8503} C_DIS
LIN {X 104.7791,Y 35.7823,Z 111,A 15.1222,B 24.9354,C -1.8569,E1 25.1506,E2 430.575} C_DIS
LIN {X 103.2435,Y 39.9986,Z 111,A 17.252,B 24.9354,C -1.8551,E1 25.1485,E2 428.4614} C_DIS
LIN {X 102.1052,Y 42.8182,Z 111,A 18.814,B 24.9352,C -1.8591,E1 25.1469,E2 426.8983} C_DIS
LIN {X 100.8251,Y 45.7519,Z 111,A 20.7191,B 24.9341,C -1.8751,E1 25.1447,E2 424.9659} C_DIS
LIN {X 98.7291,Y 50.1148,Z 111,A 22.9834,B 24.9344,C -1.8713,E1 25.1419,E2 422.7226} C_DIS
LIN {X 96.9418,Y 53.4925,Z 111,A 25.1712,B 24.9333,C -1.8862,E1 25.1389,E2 420.5112} C_DIS
LIN {X 94.5829,Y 57.5579,Z 111,A 27.3111,B 24.9338,C -1.8796,E1 25.1359,E2 418.3978} C_DIS
LIN {X 92.3545,Y 61.0697,Z 111,A 30.4112,B 24.9303,C -1.9279,E1 25.131,E2 415.1993} C_DIS
LIN {X 88.9976,Y 65.8681,Z 111,A 32.3667,B 24.9332,C -1.8872,E1 25.128,E2 413.3493} C_DIS
LIN {X 87.1376,Y 68.3086,Z 111,A 34.1005,B 24.9325,C -1.8975,E1 25.125,E2 411.5993} C_DIS
LIN {X 84.8658,Y 71.1115,Z 111,A 36.0037,B 24.9321,C -1.9036,E1 25.1216,E2 409.6906} C_DIS
LIN {X 82.6692,Y 73.6526,Z 111,A 37.7197,B 24.9319,C -1.9066,E1 25.1184,E2 407.9751} C_DIS
LIN {X 79.8525,Y 76.6972,Z 111,A 39.7917,B 24.9317,C -1.9081,E1 25.1145,E2 405.9087} C_DIS
LIN {X 77.0804,Y 79.4831,Z 111,A 41.7938,B 24.9315,C -1.911,E1 25.1105,E2 403.9081} C_DIS
LIN {X 74.7061,Y 81.7183,Z 111,A 43.469,B 24.9313,C -1.9139,E1 25.1071,E2 402.2328} C_DIS
LIN {X 71.2152,Y 84.7796,Z 111,A 47.0612,B 24.9271,C -1.9712,E1 25.0992,E2 398.519} C_DIS
LIN {X 65.8791,Y 88.9893,Z 111,A 49.2778,B 24.9309,C -1.9201,E1 25.0945,E2 396.4312} C_DIS
LIN {X 62.6621,Y 91.2837,Z 111,A 51.3879,B 24.9304,C -1.9264,E1 25.0897,E2 394.3135} C_DIS
LIN {X 59.7905,Y 93.1877,Z 111,A 53.1877,B 24.9302,C -1.9301,E1 25.0854,E2 392.5111} C_DIS
LIN {X 57.3561,Y 94.7056,Z 111,A 55.0089,B 24.9289,C -1.9469,E1 25.081,E2 390.6557} C_DIS
LIN {X 54.5271,Y 96.3641,Z 111,A 56.4502,B 24.9296,C -1.9382,E1 25.0776,E2 389.2392} C_DIS
LIN {X 51.2336,Y 98.1536,Z 111,A 58.3474,B 24.9296,C -1.939,E1 25.0729,E2 387.3456} C_DIS
LIN {X 48.162,Y 99.6961,Z 111,A 60.2384,B 24.929,C -1.9461,E1 25.0681,E2 385.4428} C_DIS
LIN {X 44.8715,Y 101.2218,Z 111,A 62.0558,B 24.929,C -1.9457,E1 25.0635,E2 383.631} C_DIS
LIN {X 41.7464,Y 102.548,Z 111,A 64.194,B 24.9277,C -1.9639,E1 25.0579,E2 381.4545} C_DIS
LIN {X 38.1449,Y 103.9416,Z 111,A 66.1102,B 24.9278,C -1.9623,E1 25.0529,E2 379.5462} C_DIS
LIN {X 34.7523,Y 105.1259,Z 111,A 67.5026,B 24.9292,C -1.9438,E1 25.0493,E2 378.2001} C_DIS
LIN {X 32.4805,Y 105.8488,Z 111,A 68.8099,B 24.9289,C -1.9479,E1 25.0458,E2 376.8856} C_DIS
LIN {X 29.0988,Y 106.8277,Z 111,A 70.6451,B 24.9287,C -1.9497,E1 25.0409,E2 375.049} C_DIS
LIN {X 25.3398,Y 107.7818,Z 111,A 72.5612,B 24.9289,C -1.9471,E1 25.0357,E2 373.1421} C_DIS
LIN {X 22.6425,Y 108.3804,Z 111,A 73.9857,B 24.9289,C -1.9475,E1 25.0318,E2 371.7184} C_DIS
LIN {X 18.9197,Y 109.0931,Z 111,A 76.0462,B 24.9285,C -1.9524,E1 25.0261,E2 369.6485} C_DIS
LIN {X 14.895,Y 109.7152,Z 111,A 78.2022,B 24.9283,C -1.955,E1 25.0202,E2 367.4883} C_DIS
LIN {X 11.1232,Y 110.1603,Z 111,A 80.1162,B 24.9285,C -1.9532,E1 25.0149,E2 365.5799} C_DIS
LIN {X 7.4473,Y 110.4689,Z 111,A 81.9109,B 24.9288,C -1.9486,E1 25.0099,E2 363.7972} C_DIS
LIN {X 4.3486,Y 110.635,Z 111,A 83.5076,B 24.9288,C -1.9481,E1 25.0055,E2 362.202} C_DIS
LIN {X 0.9195,Y 110.7161,Z 111,A 85.3235,B 24.9288,C -1.9496,E1 25.0004,E2 360.3829} C_DIS
LIN {X -2.0418,Y 110.7008,Z 111,A 86.9015,B 24.9286,C -1.9511,E1 24.996,E2 358.8013} C_DIS
LIN {X -5.9807,Y 110.5581,Z 111,A 88.8988,B 24.9288,C -1.9486,E1 24.9904,E2 356.8093} C_DIS
LIN {X -9.2007,Y 110.3374,Z 111,A 90.617,B 24.9288,C -1.9499,E1 24.9856,E2 355.0874} C_DIS
LIN {X -12.6305,Y 109.9972,Z 111,A 92.3582,B 24.9289,C -1.9472,E1 24.9808,E2 353.3516} C_DIS
LIN {X -15.5832,Y 109.6175,Z 111,A 93.7737,B 24.9294,C -1.9411,E1 24.9769,E2 351.9495} C_DIS
LIN {X -19.1667,Y 109.0489,Z 111,A 95.7305,B 24.9292,C -1.9429,E1 24.9715,E2 349.9864} C_DIS
LIN {X -22.0548,Y 108.501,Z 111,A 97.2809,B 24.9292,C -1.9429,E1 24.9672,E2 348.4344} C_DIS
LIN {X -25.2746,Y 107.7969,Z 111,A 98.9747,B 24.9294,C -1.9409,E1 24.9626,E2 346.7432} C_DIS
LIN {X -28.5889,Y 106.9654,Z 111,A 100.7727,B 24.9294,C -1.9403,E1 24.9578,E2 344.9439} C_DIS
LIN {X -30.9912,Y 106.2951,Z 111,A 102.4285,B 24.9284,C -1.9537,E1 24.9533,E2 343.2536} C_DIS
LIN {X -35.6317,Y 104.8298,Z 111,A 104.5283,B 24.9299,C -1.9338,E1 24.9478,E2 341.1974} C_DIS
LIN {X -38.7951,Y 103.7014,Z 111,A 106.3916,B 24.9297,C -1.9366,E1 24.9429,E2 339.3237} C_DIS
LIN {X -42.2628,Y 102.3378,Z 111,A 108.4022,B 24.9297,C -1.9372,E1 24.9376,E2 337.3072} C_DIS
LIN {X -45.7714,Y 100.8162,Z 111,A 111.168,B 24.9275,C -1.9659,E1 24.9304,E2 334.4662} C_DIS
LIN {X -50.6604,Y 98.4503,Z 111,A 112.9313,B 24.9309,C -1.9193,E1 24.9263,E2 332.8092} C_DIS
LIN {X -54.3687,Y 96.4525,Z 111,A 115.3839,B 24.9304,C -1.9263,E1 24.9202,E2 330.3328} C_DIS
LIN {X -56.9497,Y 94.9526,Z 111,A 116.9892,B 24.9304,C -1.9259,E1 24.9164,E2 328.7236} C_DIS
LIN {X -62.1593,Y 91.6247,Z 111,A 120.6653,B 24.9295,C -1.9387,E1 24.9077,E2 325.005} C_DIS
LIN {X -65.6566,Y 89.1524,Z 111,A 122.4137,B 24.9312,C -1.9155,E1 24.9039,E2 323.3057} C_DIS
LIN {X -69.4371,Y 86.2407,Z 111,A 124.8795,B 24.9316,C -1.91,E1 24.8985,E2 320.8438} C_DIS
LIN {X -72.395,Y 83.7743,Z 111,A 126.8479,B 24.932,C -1.9045,E1 24.8943,E2 318.8808} C_DIS
LIN {X -75.1965,Y 81.2683,Z 111,A 128.523,B 24.9331,C -1.8895,E1 24.8909,E2 317.2349} C_DIS
LIN {X -77.8931,Y 78.6863,Z 111,A 130.9211,B 24.9321,C -1.9031,E1 24.886,E2 314.7944} C_DIS
LIN {X -80.9958,Y 75.4902,Z 111,A 133.0452,B 24.933,C -1.8902,E1 24.882,E2 312.6916} C_DIS
LIN {X -83.7259,Y 72.4505,Z 111,A 135.8984,B 24.9313,C -1.9138,E1 24.8766,E2 309.7694} C_DIS
LIN {X -86.8969,Y 68.6133,Z 111,A 137.2745,B 24.9351,C -1.8602,E1 24.8744,E2 308.5147} C_DIS
LIN {X -89.9771,Y 64.5216,Z 111,A 140.2972,B 24.9346,C -1.8673,E1 24.8693,E2 305.4605} C_DIS
LIN {X -91.9008,Y 61.7514,Z 111,A 142.1753,B 24.9346,C -1.8675,E1 24.8663,E2 303.5724} C_DIS
LIN {X -93.858,Y 58.7326,Z 111,A 143.9538,B 24.9352,C -1.859,E1 24.8637,E2 301.8051} C_DIS
LIN {X -95.9102,Y 55.3182,Z 111,A 146.0963,B 24.9354,C -1.8562,E1 24.8606,E2 299.6584} C_DIS
LIN {X -97.577,Y 52.3245,Z 111,A 147.819,B 24.9359,C -1.849,E1 24.8583,E2 297.9437} C_DIS
LIN {X -99.1523,Y 49.2714,Z 111,A 149.3944,B 24.9368,C -1.836,E1 24.8564,E2 296.3909} C_DIS
LIN {X -100.8989,Y 45.5881,Z 111,A 151.7811,B 24.9365,C -1.8402,E1 24.8535,E2 293.981} C_DIS
LIN {X -102.3868,Y 42.1422,Z 111,A 153.5257,B 24.9375,C -1.8267,E1 24.8516,E2 292.2591} C_DIS
LIN {X -103.8916,Y 38.2821,Z 111,A 155.8865,B 24.9373,C -1.8284,E1 24.8493,E2 289.8811} C_DIS
LIN {X -105.0604,Y 34.9479,Z 111,A 157.6728,B 24.9378,C -1.821,E1 24.8477,E2 288.1021} C_DIS
LIN {X -106.6775,Y 29.6491,Z 111,A 160.5107,B 24.9385,C -1.8108,E1 24.8454,E2 285.2722} C_DIS
LIN {X -107.8569,Y 25.0146,Z 111,A 163.067,B 24.9389,C -1.806,E1 24.8437,E2 282.7123} C_DIS
LIN {X -108.8047,Y 20.5078,Z 111,A 165.6169,B 24.9389,C -1.8048,E1 24.8423,E2 280.1504} C_DIS
LIN {X -109.4355,Y 16.8144,Z 111,A 167.4372,B 24.9397,C -1.7939,E1 24.8415,E2 278.345} C_DIS
LIN {X -109.9402,Y 13.117,Z 111,A 169.4542,B 24.9399,C -1.791,E1 24.8408,E2 276.3231} C_DIS
LIN {X -110.2517,Y 10.1691,Z 111,A 170.9416,B 24.9403,C -1.7842,E1 24.8404,E2 274.8428} C_DIS
LIN {X -110.5343,Y 6.4109,Z 111,A 172.6481,B 24.9414,C -1.7686,E1 24.84,E2 273.1634} C_DIS
LIN {X -110.6528,Y 3.8759,Z 111,A 174.3109,B 24.9408,C -1.7777,E1 24.8398,E2 271.4689} C_DIS
LIN {X -110.7226,Y -0.0123,Z 111,A 176.3609,B 24.9411,C -1.7726,E1 24.8398,E2 269.4188} C_DIS
LIN {X -110.6655,Y -3.4631,Z 111,A 178.1178,B 24.9416,C -1.7657,E1 24.8399,E2 267.6676} C_DIS
LIN {X -110.4598,Y -7.5822,Z 111,A -179.7768,B 24.9421,C -1.7577,E1 24.8403,E2 265.5685} C_DIS
LIN {X -110.1464,Y -11.2557,Z 111,A -177.8937,B 24.9426,C -1.7507,E1 24.8407,E2 263.6911} C_DIS
LIN {X -109.6185,Y -15.5763,Z 111,A -175.6001,B 24.9429,C -1.7451,E1 24.8416,E2 261.397} C_DIS
LIN {X -108.7007,Y -21.0477,Z 111,A -172.5985,B 24.9432,C -1.7411,E1 24.843,E2 258.3873} C_DIS
LIN {X -107.7454,Y -25.4975,Z 111,A -170.214,B 24.9436,C -1.7348,E1 24.8445,E2 256.0036} C_DIS
LIN {X -106.8434,Y -29.0406,Z 111,A -168.381,B 24.9441,C -1.7268,E1 24.8458,E2 254.1791} C_DIS
LIN {X -105.7727,Y -32.726,Z 111,A -166.4623,B 24.9447,C -1.7181,E1 24.8473,E2 252.27} C_DIS
LIN {X -104.7307,Y -35.9256,Z 111,A -164.6299,B 24.9447,C -1.7164,E1 24.849,E2 250.4313} C_DIS
LIN {X -103.5567,Y -39.1772,Z 111,A -162.9668,B 24.9454,C -1.7062,E1 24.8506,E2 248.783} C_DIS
LIN {X -102.0356,Y -42.9835,Z 111,A -160.7407,B 24.9456,C -1.7041,E1 24.8529,E2 246.5495} C_DIS
LIN {X -100.5179,Y -46.4232,Z 111,A -158.8627,B 24.9461,C -1.6959,E1 24.8551,E2 244.6807} C_DIS
LIN {X -98.9559,Y -49.6677,Z 111,A -156.8703,B 24.9461,C -1.6957,E1 24.8575,E2 242.6781} C_DIS
LIN {X -97.3617,Y -52.7214,Z 111,A -155.1349,B 24.9465,C -1.6889,E1 24.8598,E2 240.9496} C_DIS
LIN {X -95.635,Y -55.796,Z 111,A -153.3936,B 24.9471,C -1.6807,E1 24.8622,E2 239.2188} C_DIS
LIN {X -94.1662,Y -58.2392,Z 111,A -151.7436,B 24.9469,C -1.6837,E1 24.8646,E2 237.5534} C_DIS
LIN {X -92.1972,Y -61.3083,Z 111,A -149.7875,B 24.947,C -1.6815,E1 24.8676,E2 235.5925} C_DIS
LIN {X -90.0164,Y -64.4665,Z 111,A -147.9173,B 24.9476,C -1.6719,E1 24.8706,E2 233.736} C_DIS
LIN {X -88.0086,Y -67.1832,Z 111,A -146.1079,B 24.9477,C -1.6701,E1 24.8737,E2 231.9224} C_DIS
LIN {X -85.9986,Y -69.7358,Z 111,A -144.4771,B 24.9481,C -1.6641,E1 24.8765,E2 230.2982} C_DIS
LIN {X -83.9261,Y -72.2188,Z 111,A -142.7516,B 24.9482,C -1.6622,E1 24.8796,E2 228.5693} C_DIS
LIN {X -80.9724,Y -75.515,Z 111,A -140.4364,B 24.9485,C -1.6581,E1 24.884,E2 226.2537} C_DIS
LIN {X -78.884,Y -77.6929,Z 111,A -139.0013,B 24.949,C -1.6497,E1 24.8867,E2 224.8324} C_DIS
LIN {X -76.6495,Y -79.8984,Z 111,A -137.3352,B 24.9491,C -1.6479,E1 24.8901,E2 223.1636} C_DIS
LIN {X -74.2154,Y -82.1654,Z 111,A -135.4995,B 24.9491,C -1.649,E1 24.8939,E2 221.3179} C_DIS
LIN {X -71.3948,Y -84.6281,Z 111,A -133.5623,B 24.9493,C -1.6452,E1 24.898,E2 219.3822} C_DIS
LIN {X -68.59,Y -86.9152,Z 111,A -131.6504,B 24.9493,C -1.6433,E1 24.9022,E2 217.4675} C_DIS
LIN {X -65.3839,Y -89.352,Z 111,A -129.5825,B 24.9497,C -1.639,E1 24.9068,E2 215.4026} C_DIS
LIN {X -62.3144,Y -91.5196,Z 111,A -127.7249,B 24.9501,C -1.6323,E1 24.911,E2 213.5547} C_DIS
LIN {X -59.8375,Y -93.1575,Z 111,A -125.5381,B 24.9486,C -1.6563,E1 24.9163,E2 211.3035} C_DIS
LIN {X -56.2228,Y -95.3827,Z 111,A -123.9074,B 24.9502,C -1.63,E1 24.9201,E2 209.7305} C_DIS
LIN {X -52.7823,Y -97.3287,Z 111,A -122.1014,B 24.951,C -1.6174,E1 24.9244,E2 207.9492} C_DIS
LIN {X -50.0358,Y -98.7695,Z 111,A -120.2682,B 24.9505,C -1.6246,E1 24.929,E2 206.0938} C_DIS
LIN {X -46.8183,Y -100.334,Z 111,A -118.5301,B 24.951,C -1.6178,E1 24.9334,E2 204.3675} C_DIS
LIN {X -44.6892,Y -101.3013,Z 111,A -115.8353,B 24.9472,C -1.6781,E1 24.9407,E2 201.5231} C_DIS
LIN {X -37.7454,Y -104.0873,Z 111,A -113.3711,B 24.9511,C -1.6157,E1 24.9468,E2 199.202} C_DIS
LIN {X -34.0269,Y -105.3614,Z 111,A -111.3129,B 24.9511,C -1.6151,E1 24.9522,E2 197.1415} C_DIS
LIN {X -30.4819,Y -106.4415,Z 111,A -109.3755,B 24.9511,C -1.6145,E1 24.9574,E2 195.2021} C_DIS
LIN {X -27.5485,Y -107.2377,Z 111,A -107.7891,B 24.9511,C -1.6141,E1 24.9617,E2 193.6143} C_DIS
LIN {X -23.8926,Y -108.1114,Z 111,A -105.781,B 24.9511,C -1.6158,E1 24.9672,E2 191.5996} C_DIS
LIN {X -20.2222,Y -108.8591,Z 111,A -103.7529,B 24.9509,C -1.6188,E1 24.9727,E2 189.5622} C_DIS
LIN {X -16.4285,Y -109.4952,Z 111,A -101.8485,B 24.9512,C -1.6146,E1 24.978,E2 187.666} C_DIS
LIN {X -12.9483,Y -109.9599,Z 111,A -100.0166,B 24.9512,C -1.615,E1 24.9831,E2 185.8321} C_DIS
LIN {X -9.1919,Y -110.3381,Z 111,A -98.0753,B 24.9512,C -1.6143,E1 24.9885,E2 183.8913} C_DIS
LIN {X -5.5032,Y -110.5845,Z 111,A -96.1547,B 24.9512,C -1.6147,E1 24.9938,E2 181.9692} C_DIS
LIN {X -1.9868,Y -110.7018,Z 111,A -94.4206,B 24.9514,C -1.6113,E1 24.9986,E2 180.243} C_DIS
LIN {X 0.7699,Y -110.7126,Z 111,A -93.3494,B 24.9522,C -1.5966,E1 25.0015,E2 179.2066} C_DIS
Enddeposition()
LIN {X 0.7699,Y -110.7126,Z 111,A -93.3494,B 24.9522,C -1.5966,E1 25.0015,E2 179.2066} C_DIS
Startdeposition()
$VEL.CP = VEL_PRINT
LIN {X -1.4499,Y -109.7742,Z 111,A -95.0315,B 24.9526,C -1.5909,E1 24.9968,E2 180.9024} C_DIS
LIN {X -4.9617,Y -109.6704,Z 111,A -96.8571,B 24.9526,C -1.591,E1 24.9917,E2 182.7279} C_DIS
LIN {X -8.7017,Y -109.4369,Z 111,A -98.7509,B 24.9524,C -1.5936,E1 24.9864,E2 184.6164} C_DIS
LIN {X -12.4671,Y -109.0726,Z 111,A -100.7341,B 24.9524,C -1.5934,E1 24.9809,E2 186.6011} C_DIS
LIN {X -15.9163,Y -108.6235,Z 111,A -102.5671,B 24.9524,C -1.5931,E1 24.9758,E2 188.4364} C_DIS
LIN {X -20.0063,Y -107.9456,Z 111,A -104.6358,B 24.9522,C -1.5976,E1 24.9702,E2 190.4963} C_DIS
LIN {X -24.6656,Y -106.9755,Z 111,A -107.1861,B 24.9522,C -1.5961,E1 24.9632,E2 193.0533} C_DIS
LIN {X -27.9247,Y -106.1732,Z 111,A -109.0373,B 24.9525,C -1.593,E1 24.9582,E2 194.9145} C_DIS
LIN {X -31.6316,Y -105.1274,Z 111,A -111.2586,B 24.9529,C -1.5859,E1 24.9522,E2 197.1564} C_DIS
LIN {X -35.3693,Y -103.9292,Z 111,A -113.0644,B 24.9522,C -1.5973,E1 24.9474,E2 198.9384} C_DIS
LIN {X -40.0139,Y -102.2304,Z 111,A -116.1367,B 24.9532,C -1.5801,E1 24.9393,E2 202.058} C_DIS
LIN {X -43.638,Y -100.737,Z 111,A -117.4821,B 24.9514,C -1.6102,E1 24.936,E2 203.3351} C_DIS
LIN {X -46.6569,Y -99.3752,Z 111,A -119.3113,B 24.9515,C -1.6081,E1 24.9313,E2 205.1737} C_DIS
LIN {X -49.1179,Y -98.1823,Z 111,A -121.2169,B 24.9526,C -1.5909,E1 24.9265,E2 207.1253} C_DIS
LIN {X -52.0687,Y -96.6494,Z 111,A -122.6353,B 24.9517,C -1.6057,E1 24.923,E2 208.5123} C_DIS
LIN {X -58.7844,Y -92.7196,Z 111,A -126.7349,B 24.9514,C -1.6101,E1 24.9132,E2 212.6141} C_DIS
LIN {X -62.1544,Y -90.4951,Z 111,A -128.6435,B 24.9507,C -1.6214,E1 24.9088,E2 214.5022} C_DIS
LIN {X -64.4774,Y -88.854,Z 111,A -130.3985,B 24.9512,C -1.6133,E1 24.9048,E2 216.2825} C_DIS
LIN {X -69.1601,Y -85.2587,Z 111,A -133.1792,B 24.9502,C -1.6307,E1 24.8987,E2 219.0321} C_DIS
LIN {X -71.3077,Y -83.4709,Z 111,A -134.8436,B 24.9505,C -1.6254,E1 24.8951,E2 220.7154} C_DIS
LIN {X -74.0661,Y -81.0335,Z 111,A -136.735,B 24.9502,C -1.6304,E1 24.8912,E2 222.6026} C_DIS
LIN {X -76.5716,Y -78.6717,Z 111,A -138.6138,B 24.9502,C -1.6309,E1 24.8874,E2 224.4878} C_DIS
LIN {X -79.1104,Y -76.1164,Z 111,A -140.4089,B 24.9497,C -1.6383,E1 24.8839,E2 226.2731} C_DIS
LIN {X -82.6052,Y -72.3087,Z 111,A -143.1128,B 24.9493,C -1.6441,E1 24.8789,E2 228.9751} C_DIS
LIN {X -84.8535,Y -69.6596,Z 111,A -145.0941,B 24.9495,C -1.6419,E1 24.8753,E2 230.9709} C_DIS
LIN {X -87.3265,Y -66.5325,Z 111,A -147.1097,B 24.949,C -1.6494,E1 24.8719,E2 232.9781} C_DIS
LIN {X -89.3007,Y -63.8557,Z 111,A -148.7744,B 24.9486,C -1.6565,E1 24.8691,E2 234.634} C_DIS
LIN {X -91.8486,Y -60.1342,Z 111,A -151.1637,B 24.9483,C -1.6612,E1 24.8654,E2 237.0242} C_DIS
LIN {X -94.3855,Y -56.0677,Z 111,A -153.6585,B 24.9479,C -1.668,E1 24.8618,E2 239.5153} C_DIS
LIN {X -96.0071,Y -53.2437,Z 111,A -155.4117,B 24.9477,C -1.6706,E1 24.8594,E2 241.2716} C_DIS
LIN {X -97.7426,Y -49.9855,Z 111,A -157.3292,B 24.9473,C -1.6763,E1 24.8569,E2 243.1858} C_DIS
LIN {X -99.7759,Y -45.796,Z 111,A -159.6575,B 24.9467,C -1.687,E1 24.8541,E2 245.5012} C_DIS
LIN {X -100.9116,Y -43.2369,Z 111,A -161.5618,B 24.9475,C -1.6745,E1 24.852,E2 247.4459} C_DIS
LIN {X -102.8042,Y -38.5177,Z 111,A -164.004,B 24.9465,C -1.6902,E1 24.8495,E2 249.8642} C_DIS
LIN {X -104.0245,Y -35.0864,Z 111,A -165.7831,B 24.9458,C -1.7005,E1 24.8479,E2 251.6288} C_DIS
LIN {X -104.895,Y -32.3915,Z 111,A -167.2845,B 24.9456,C -1.7041,E1 24.8466,E2 253.1303} C_DIS
LIN {X -105.8722,Y -29.0415,Z 111,A -169.1791,B 24.9454,C -1.7069,E1 24.8452,E2 255.0293} C_DIS
LIN {X -106.7289,Y -25.7137,Z 111,A -171.0368,B 24.9452,C -1.71,E1 24.8439,E2 256.8903} C_DIS
LIN {X -107.5861,Y -21.8506,Z 111,A -173.7868,B 24.9464,C -1.691,E1 24.8424,E2 259.7019} C_DIS
LIN {X -108.4463,Y -17.0779,Z 111,A -176.4055,B 24.9461,C -1.6958,E1 24.8412,E2 262.3249} C_DIS
LIN {X -109.1307,Y -11.955,Z 111,A -178.1435,B 24.9433,C -1.74,E1 24.8407,E2 263.9677} C_DIS
LIN {X -109.4235,Y -8.8698,Z 111,A -179.9103,B 24.9433,C -1.7396,E1 24.8402,E2 265.7461} C_DIS
LIN {X -109.7035,Y -4.1875,Z 111,A 177.2114,B 24.9438,C -1.7315,E1 24.8398,E2 268.6612} C_DIS
LIN {X -109.7795,Y -0.8703,Z 111,A 176.1112,B 24.9419,C -1.7606,E1 24.8398,E2 269.6984} C_DIS
LIN {X -109.7598,Y 2.2339,Z 111,A 173.7001,B 24.9435,C -1.7364,E1 24.8399,E2 272.1819} C_DIS
LIN {X -109.6106,Y 6.1389,Z 111,A 172.2225,B 24.9417,C -1.7639,E1 24.8401,E2 273.6027} C_DIS
LIN {X -109.1816,Y 11.4686,Z 111,A 169.3675,B 24.9412,C -1.7705,E1 24.8408,E2 276.459} C_DIS
LIN {X -108.7051,Y 15.3421,Z 111,A 167.3235,B 24.9408,C -1.7769,E1 24.8415,E2 278.5002} C_DIS
LIN {X -108.1281,Y 18.9915,Z 111,A 164.9911,B 24.9414,C -1.768,E1 24.8426,E2 280.8675} C_DIS
LIN {X -107.52,Y 22.1727,Z 111,A 163.7562,B 24.9399,C -1.7904,E1 24.8433,E2 282.0563} C_DIS
LIN {X -106.8224,Y 25.3285,Z 111,A 161.611,B 24.9407,C -1.7787,E1 24.8447,E2 284.242} C_DIS
LIN {X -105.2599,Y 31.185,Z 111,A 158.7612,B 24.9392,C -1.8005,E1 24.8468,E2 287.0565} C_DIS
LIN {X -103.9213,Y 35.3925,Z 111,A 156.444,B 24.9388,C -1.8072,E1 24.8488,E2 289.3708} C_DIS
LIN {X -101.3422,Y 42.2151,Z 111,A 152.8245,B 24.9375,C -1.826,E1 24.8524,E2 292.966} C_DIS
LIN {X -98.7864,Y 47.891,Z 111,A 149.329,B 24.9375,C -1.8265,E1 24.8565,E2 296.4792} C_DIS
LIN {X -97.2745,Y 50.8913,Z 111,A 147.5053,B 24.9373,C -1.8291,E1 24.8588,E2 298.3065} C_DIS
LIN {X -95.35,Y 54.4117,Z 111,A 145.1171,B 24.9376,C -1.8242,E1 24.8621,E2 300.719} C_DIS
LIN {X -93.6994,Y 57.2068,Z 111,A 143.8729,B 24.9361,C -1.8459,E1 24.8638,E2 301.9177} C_DIS
LIN {X -92.0353,Y 59.8505,Z 111,A 141.7624,B 24.9371,C -1.8325,E1 24.8671,E2 304.0709} C_DIS
LIN {X -88.6351,Y 64.7765,Z 111,A 138.5206,B 24.9368,C -1.8367,E1 24.8724,E2 307.3186} C_DIS
LIN {X -86.3693,Y 67.7691,Z 111,A 136.8485,B 24.9357,C -1.8527,E1 24.8752,E2 308.9605} C_DIS
LIN {X -83.0191,Y 71.8348,Z 111,A 134.433,B 24.9343,C -1.8725,E1 24.8795,E2 311.3399} C_DIS
LIN {X -80.3427,Y 74.8154,Z 111,A 132.0005,B 24.9348,C -1.8648,E1 24.8841,E2 313.8015} C_DIS
LIN {X -76.8056,Y 78.4424,Z 111,A 129.1699,B 24.9348,C -1.8642,E1 24.8897,E2 316.6456} C_DIS
LIN {X -71.9139,Y 82.9486,Z 111,A 125.8354,B 24.9339,C -1.8774,E1 24.8966,E2 319.9618} C_DIS
LIN {X -68.3875,Y 85.8798,Z 111,A 123.4803,B 24.9335,C -1.8841,E1 24.9017,E2 322.3099} C_DIS
LIN {X -65.4317,Y 88.1547,Z 111,A 121.5108,B 24.9332,C -1.8873,E1 24.9061,E2 324.2789} C_DIS
LIN {X -58.9217,Y 92.6315,Z 111,A 118.0735,B 24.9307,C -1.922,E1 24.9138,E2 327.6452} C_DIS
LIN {X -54.319,Y 95.4033,Z 111,A 114.4961,B 24.9325,C -1.8971,E1 24.9226,E2 331.2926} C_DIS
LIN {X -50.3827,Y 97.5395,Z 111,A 112.2814,B 24.9319,C -1.9058,E1 24.928,E2 333.4929} C_DIS
LIN {X -45.1971,Y 100.0469,Z 111,A 109.3439,B 24.9314,C -1.9132,E1 24.9354,E2 336.4202} C_DIS
LIN {X -41.9001,Y 101.4734,Z 111,A 107.3535,B 24.9315,C -1.9114,E1 24.9405,E2 338.4196} C_DIS
LIN {X -37.3227,Y 103.2437,Z 111,A 104.8637,B 24.9311,C -1.9176,E1 24.947,E2 340.8997} C_DIS
LIN {X -33.7736,Y 104.4581,Z 111,A 101.9243,B 24.9336,C -1.8817,E1 24.9551,E2 343.9297} C_DIS
LIN {X -28.0705,Y 106.1345,Z 111,A 99.7372,B 24.9308,C -1.9206,E1 24.9607,E2 346.0278} C_DIS
LIN {X -24.5976,Y 106.9913,Z 111,A 97.9497,B 24.9305,C -1.9255,E1 24.9655,E2 347.8061} C_DIS
LIN {X -20.441,Y 107.863,Z 111,A 95.4379,B 24.9312,C -1.9157,E1 24.9725,E2 350.3441} C_DIS
LIN {X -15.3084,Y 108.7098,Z 111,A 93.1426,B 24.9299,C -1.9343,E1 24.9787,E2 352.5973} C_DIS
LIN {X -12.3964,Y 109.0808,Z 111,A 91.5198,B 24.9301,C -1.9315,E1 24.9832,E2 354.2277} C_DIS
LIN {X -8.8843,Y 109.4223,Z 111,A 89.6519,B 24.9301,C -1.9314,E1 24.9884,E2 356.0969} C_DIS
LIN {X -5.9364,Y 109.6218,Z 111,A 87.8206,B 24.9309,C -1.9204,E1 24.9936,E2 357.9549} C_DIS
LIN {X -1.3258,Y 109.7762,Z 111,A 85.6007,B 24.9303,C -1.9285,E1 24.9997,E2 360.1556} C_DIS
LIN {X 1.9307,Y 109.7654,Z 111,A 83.9591,B 24.9301,C -1.9312,E1 25.0043,E2 361.7908} C_DIS
LIN {X 5.8049,Y 109.629,Z 111,A 81.9527,B 24.9301,C -1.9319,E1 25.0099,E2 363.7948} C_DIS
LIN {X 9.321,Y 109.3874,Z 111,A 80.023,B 24.9303,C -1.9282,E1 25.0153,E2 365.7325} C_DIS
LIN {X 12.7864,Y 109.0352,Z 111,A 78.3128,B 24.93,C -1.9323,E1 25.02,E2 367.4317} C_DIS
LIN {X 16.9407,Y 108.4675,Z 111,A 76.1307,B 24.93,C -1.9319,E1 25.026,E2 369.6126} C_DIS
LIN {X 21.9419,Y 107.5673,Z 111,A 73.7949,B 24.9292,C -1.9439,E1 25.0324,E2 371.9175} C_DIS
LIN {X 24.5222,Y 107.0087,Z 111,A 72.099,B 24.9302,C -1.9301,E1 25.0371,E2 373.6439} C_DIS
LIN {X 28.1792,Y 106.1052,Z 111,A 69.6662,B 24.9316,C -1.9096,E1 25.0438,E2 376.1213} C_DIS
LIN {X 31.6272,Y 105.1287,Z 111,A 68.3816,B 24.93,C -1.9324,E1 25.0471,E2 377.3498} C_DIS
LIN {X 34.3289,Y 104.2785,Z 111,A 66.4535,B 24.9314,C -1.9126,E1 25.0523,E2 379.3213} C_DIS
LIN {X 40.7626,Y 101.9363,Z 111,A 63.2909,B 24.9304,C -1.9263,E1 25.0605,E2 382.4447} C_DIS
LIN {X 43.9913,Y 100.583,Z 111,A 61.4061,B 24.9308,C -1.9219,E1 25.0653,E2 384.3354} C_DIS
LIN {X 49.3794,Y 98.0523,Z 111,A 58.3793,B 24.9308,C -1.9214,E1 25.0729,E2 387.3554} C_DIS
LIN {X 56.1312,Y 94.348,Z 111,A 54.3313,B 24.9313,C -1.9145,E1 25.0828,E2 391.4078} C_DIS
LIN {X 59.3711,Y 92.343,Z 111,A 52.4277,B 24.9313,C -1.9151,E1 25.0873,E2 393.3042} C_DIS
LIN {X 61.7132,Y 90.7947,Z 111,A 50.7948,B 24.9319,C -1.9055,E1 25.0911,E2 394.9541} C_DIS
LIN {X 65.4125,Y 88.1691,Z 111,A 48.1514,B 24.9331,C -1.8897,E1 25.0972,E2 397.6257} C_DIS
LIN {X 70.5407,Y 84.1213,Z 111,A 45.0837,B 24.9325,C -1.8979,E1 25.1038,E2 400.6624} C_DIS
LIN {X 73.2596,Y 81.763,Z 111,A 43.2288,B 24.9327,C -1.8951,E1 25.1077,E2 402.5164} C_DIS
LIN {X 76.0263,Y 79.1972,Z 111,A 41.2712,B 24.9329,C -1.8916,E1 25.1116,E2 404.4745} C_DIS
LIN {X 78.3638,Y 76.8857,Z 111,A 39.4508,B 24.9335,C -1.8833,E1 25.1152,E2 406.3065} C_DIS
LIN {X 80.959,Y 74.1472,Z 111,A 37.5869,B 24.9335,C -1.8835,E1 25.1188,E2 408.1619} C_DIS
LIN {X 83.4721,Y 71.3063,Z 111,A 35.6313,B 24.9337,C -1.88,E1 25.1224,E2 410.117} C_DIS
LIN {X 85.7212,Y 68.5889,Z 111,A 33.6629,B 24.9344,C -1.87,E1 25.1259,E2 412.0998} C_DIS
LIN {X 87.7587,Y 65.9589,Z 111,A 32.0381,B 24.9344,C -1.8706,E1 25.1286,E2 413.7154} C_DIS
LIN {X 91.406,Y 60.8055,Z 111,A 28.654,B 24.9353,C -1.8583,E1 25.134,E2 417.1119} C_DIS
LIN {X 93.6685,Y 57.2577,Z 111,A 26.5605,B 24.9353,C -1.857,E1 25.1371,E2 419.1979} C_DIS
LIN {X 97.055,Y 51.308,Z 111,A 23.3603,B 24.9349,C -1.8636,E1 25.1414,E2 422.366} C_DIS
LIN {X 99.915,Y 45.4898,Z 111,A 19.8776,B 24.9359,C -1.8496,E1 25.1457,E2 425.8631} C_DIS
LIN {X 101.3655,Y 42.1599,Z 111,A 17.7022,B 24.9371,C -1.8318,E1 25.1481,E2 428.0686} C_DIS
LIN {X 102.7206,Y 38.7382,Z 111,A 15.849,B 24.9373,C -1.8291,E1 25.15,E2 429.9177} C_DIS
LIN {X 103.692,Y 36.0585,Z 111,A 14.4564,B 24.9373,C -1.8288,E1 25.1513,E2 431.3031} C_DIS
LIN {X 105.5139,Y 30.3171,Z 111,A 11.4934,B 24.9374,C -1.8273,E1 25.1538,E2 434.2531} C_DIS
LIN {X 106.7987,Y 25.4277,Z 111,A 8.7706,B 24.9382,C -1.8153,E1 25.1557,E2 436.9883} C_DIS
LIN {X 108.0943,Y 19.1795,Z 111,A 5.4386,B 24.9389,C -1.8048,E1 25.1575,E2 440.3256} C_DIS
LIN {X 108.6767,Y 15.5418,Z 111,A 3.4846,B 24.9395,C -1.7973,E1 25.1583,E2 442.2858} C_DIS
LIN {X 109.0772,Y 12.4275,Z 111,A 1.7225,B 24.9402,C -1.7866,E1 25.1589,E2 444.0628} C_DIS
LIN {X 109.4514,Y 8.5204,Z 111,A -0.1876,B 24.9402,C -1.7862,E1 25.1594,E2 445.9626} C_DIS
LIN {X 109.6758,Y 4.8371,Z 111,A -2.1052,B 24.9406,C -1.7803,E1 25.1597,E2 447.8826} C_DIS
LIN {X 109.7684,Y 1.7637,Z 111,A -3.7683,B 24.9411,C -1.7725,E1 25.1597,E2 449.5542} C_DIS
LIN {X 109.7647,Y -1.9656,Z 111,A -5.6493,B 24.9413,C -1.7691,E1 25.1597,E2 451.4321} C_DIS
LIN {X 109.6577,Y -5.2581,Z 111,A -7.4673,B 24.942,C -1.7591,E1 25.1595,E2 453.2628} C_DIS
LIN {X 109.4116,Y -9.0181,Z 111,A -9.3215,B 24.942,C -1.7577,E1 25.1591,E2 455.1093} C_DIS
LIN {X 109.0347,Y -12.79,Z 111,A -11.2578,B 24.9424,C -1.7532,E1 25.1586,E2 457.0448} C_DIS
LIN {X 108.5695,Y -16.2807,Z 111,A -13.7393,B 24.9446,C -1.7187,E1 25.1575,E2 459.593} C_DIS
LIN {X 107.8429,Y -20.5455,Z 111,A -15.3281,B 24.9432,C -1.741,E1 25.1568,E2 461.1199} C_DIS
LIN {X 107.2495,Y -23.4456,Z 111,A -16.8933,B 24.9436,C -1.7352,E1 25.1559,E2 462.6898} C_DIS
LIN {X 106.3655,Y -27.1767,Z 111,A -18.8511,B 24.9439,C -1.7307,E1 25.1546,E2 464.6469} C_DIS
LIN {X 105.1543,Y -31.5412,Z 111,A -21.181,B 24.9443,C -1.7247,E1 25.1528,E2 466.9776} C_DIS
LIN {X 103.5277,Y -36.5268,Z 111,A -23.9971,B 24.945,C -1.7125,E1 25.1503,E2 469.8064} C_DIS
LIN {X 101.9301,Y -40.778,Z 111,A -26.2033,B 24.945,C -1.7125,E1 25.1481,E2 472.0006} C_DIS
LIN {X 100.2709,Y -44.7,Z 111,A -28.9345,B 24.9469,C -1.6831,E1 25.145,E2 474.786} C_DIS
LIN {X 98.7859,Y -47.892,Z 111,A -30.3002,B 24.9459,C -1.6984,E1 25.1434,E2 476.1083} C_DIS
LIN {X 97.1321,Y -51.1615,Z 111,A -32.4934,B 24.9471,C -1.6803,E1 25.1405,E2 478.3326} C_DIS
LIN {X 94.79,Y -55.3834,Z 111,A -35.3798,B 24.9486,C -1.6568,E1 25.1364,E2 481.2595} C_DIS
LIN {X 92.501,Y -59.125,Z 111,A -37.8623,B 24.9495,C -1.6419,E1 25.1327,E2 483.7647} C_DIS
LIN {X 89.524,Y -63.5428,Z 111,A -39.7741,B 24.9476,C -1.6721,E1 25.1297,E2 485.5958} C_DIS
LIN {X 87.5047,Y -66.297,Z 111,A -41.573,B 24.948,C -1.6665,E1 25.1267,E2 487.3993} C_DIS
LIN {X 84.6183,Y -69.9427,Z 111,A -44.2284,B 24.949,C -1.65,E1 25.122,E2 490.0813} C_DIS
LIN {X 81.5314,Y -73.5183,Z 111,A -46.5064,B 24.9489,C -1.6518,E1 25.1178,E2 492.3447} C_DIS
LIN {X 78.7778,Y -76.4615,Z 111,A -48.744,B 24.9496,C -1.6407,E1 25.1135,E2 494.599} C_DIS
LIN {X 74.7865,Y -80.3709,Z 111,A -51.4203,B 24.9493,C -1.6441,E1 25.1081,E2 497.2561} C_DIS
LIN {X 72.1205,Y -82.7696,Z 111,A -53.2467,B 24.9495,C -1.6418,E1 25.1043,E2 499.0808} C_DIS
LIN {X 69.4353,Y -85.0356,Z 111,A -55.2025,B 24.9501,C -1.6323,E1 25.1001,E2 501.0514} C_DIS
LIN {X 65.2565,Y -88.2836,Z 111,A -57.7806,B 24.9499,C -1.6344,E1 25.0944,E2 503.6153} C_DIS
LIN {X 62.6633,Y -90.1414,Z 111,A -59.5038,B 24.9503,C -1.6284,E1 25.0904,E2 505.3466} C_DIS
LIN {X 59.4914,Y -92.2658,Z 111,A -61.5229,B 24.9506,C -1.6233,E1 25.0857,E2 507.371} C_DIS
LIN {X 55.4359,Y -94.7589,Z 111,A -63.8736,B 24.9506,C -1.6244,E1 25.0801,E2 509.7118} C_DIS
LIN {X 52.0263,Y -96.6721,Z 111,A -66.6739,B 24.9527,C -1.5883,E1 25.0731,E2 512.5894} C_DIS
LIN {X 47.9119,Y -98.7764,Z 111,A -68.2503,B 24.9508,C -1.62,E1 25.0693,E2 514.0866} C_DIS
LIN {X 43.5729,Y -100.7654,Z 111,A -70.7997,B 24.9512,C -1.6137,E1 25.0628,E2 516.6446} C_DIS
LIN {X 40.4582,Y -102.0559,Z 111,A -72.7086,B 24.9517,C -1.6048,E1 25.0578,E2 518.5703} C_DIS
LIN {X 36.8813,Y -103.4033,Z 111,A -74.7448,B 24.952,C -1.6003,E1 25.0525,E2 520.6127} C_DIS
LIN {X 32.9598,Y -104.7188,Z 111,A -77.1352,B 24.9528,C -1.5879,E1 25.0461,E2 523.028} C_DIS
LIN {X 28.0224,Y -106.1475,Z 111,A -79.3987,B 24.9519,C -1.6027,E1 25.0401,E2 525.2529} C_DIS
LIN {X 23.0042,Y -107.3458,Z 111,A -82.1529,B 24.9522,C -1.5975,E1 25.0326,E2 528.0155} C_DIS
LIN {X 19.3463,Y -108.0643,Z 111,A -84.0687,B 24.9522,C -1.5972,E1 25.0273,E2 529.9299} C_DIS
LIN {X 14.7772,Y -108.7853,Z 111,A -86.4303,B 24.9522,C -1.5976,E1 25.0208,E2 532.2883} C_DIS
LIN {X 11.4578,Y -109.1828,Z 111,A -88.2269,B 24.9524,C -1.5944,E1 25.0158,E2 534.0911} C_DIS
LIN {X 7.6585,Y -109.5152,Z 111,A -90.2181,B 24.9524,C -1.5934,E1 25.0102,E2 536.0836} C_DIS
LIN {X 4.1816,Y -109.7039,Z 111,A -92.0893,B 24.9526,C -1.5905,E1 25.005,E2 537.9612} C_DIS
LIN {X 0.758,Y -109.7779,Z 111,A -93.1125,B 24.9507,C -1.6219,E1 25.0024,E2 538.9098} C_DIS
Enddeposition()
LIN {X 0.758,Y -109.7779,Z 111,A -93.1125,B 24.9507,C -1.6219,E1 25.0024,E2 538.9098} C_DIS
Startdeposition()
$VEL.CP = VEL_PRINT
LIN {X 2.5013,Y -108.8174,Z 111,A -92.0286,B 24.9493,C -1.6453,E1 25.0055,E2 537.7706} C_DIS
LIN {X 6.3863,Y -108.6581,Z 111,A -90.0113,B 24.9493,C -1.6449,E1 25.0112,E2 535.7549} C_DIS
LIN {X 9.9831,Y -108.3862,Z 111,A -88.2364,B 24.9496,C -1.6407,E1 25.0161,E2 533.9911} C_DIS
LIN {X 13.324,Y -108.0284,Z 111,A -86.3025,B 24.9491,C -1.6487,E1 25.0215,E2 532.0396} C_DIS
LIN {X 19.2587,Y -107.1276,Z 111,A -83.2932,B 24.9493,C -1.6447,E1 25.0297,E2 529.0427} C_DIS
LIN {X 22.8547,Y -106.4191,Z 111,A -80.6702,B 24.9474,C -1.676,E1 25.0371,E2 526.349} C_DIS
LIN {X 27.1822,Y -105.3962,Z 111,A -79.2974,B 24.9498,C -1.637,E1 25.0406,E2 525.0705} C_DIS
LIN {X 32.1557,Y -103.9868,Z 111,A -76.2959,B 24.9489,C -1.6519,E1 25.0487,E2 522.0387} C_DIS
LIN {X 35.7691,Y -102.8002,Z 111,A -74.3285,B 24.9489,C -1.653,E1 25.0539,E2 520.0728} C_DIS
LIN {X 39.2692,Y -101.5159,Z 111,A -72.3111,B 24.9485,C -1.658,E1 25.0592,E2 518.0478} C_DIS
LIN {X 42.9784,Y -100.002,Z 111,A -69.3967,B 24.9461,C -1.696,E1 25.0669,E2 515.0503} C_DIS
LIN {X 47.6932,Y -97.8415,Z 111,A -67.3982,B 24.9478,C -1.6685,E1 25.0717,E2 513.122} C_DIS
LIN {X 53.4818,Y -94.8006,Z 111,A -63.994,B 24.9476,C -1.6729,E1 25.0801,E2 509.7174} C_DIS
LIN {X 56.0538,Y -93.3033,Z 111,A -62.133,B 24.9466,C -1.6886,E1 25.0847,E2 507.8249} C_DIS
LIN {X 58.776,Y -91.6112,Z 111,A -60.5557,B 24.9466,C -1.6871,E1 25.0883,E2 506.2562} C_DIS
LIN {X 62.8788,Y -88.8463,Z 111,A -58.392,B 24.9475,C -1.6731,E1 25.0932,E2 504.1329} C_DIS
LIN {X 67.5467,Y -85.3504,Z 111,A -54.806,B 24.9457,C -1.7023,E1 25.1013,E2 500.491} C_DIS
LIN {X 70.1662,Y -83.2121,Z 111,A -53.3578,B 24.9464,C -1.6917,E1 25.1043,E2 499.0735} C_DIS
LIN {X 72.815,Y -80.9029,Z 111,A -51.6584,B 24.9465,C -1.6894,E1 25.1079,E2 497.3862} C_DIS
LIN {X 76.4517,Y -77.475,Z 111,A -48.4288,B 24.9444,C -1.7222,E1 25.1145,E2 494.0926} C_DIS
LIN {X 79.1906,Y -74.6733,Z 111,A -46.9334,B 24.9457,C -1.7023,E1 25.1173,E2 492.6508} C_DIS
LIN {X 81.5901,Y -72.0461,Z 111,A -44.4049,B 24.9435,C -1.7362,E1 25.1221,E2 490.0536} C_DIS
LIN {X 84.3787,Y -68.7571,Z 111,A -42.8201,B 24.9451,C -1.7117,E1 25.1248,E2 488.5338} C_DIS
LIN {X 88.2133,Y -63.7658,Z 111,A -39.4476,B 24.9443,C -1.7233,E1 25.1305,E2 485.1501} C_DIS
LIN {X 91.7663,Y -58.5343,Z 111,A -35.7746,B 24.9427,C -1.7481,E1 25.1362,E2 481.4369} C_DIS
LIN {X 93.5522,Y -55.6355,Z 111,A -34.3926,B 24.9436,C -1.735,E1 25.1381,E2 480.093} C_DIS
LIN {X 95.2335,Y -52.7066,Z 111,A -31.8605,B 24.941,C -1.774,E1 25.1416,E2 477.482} C_DIS
LIN {X 97.5143,Y -48.3548,Z 111,A -29.3416,B 24.9407,C -1.7787,E1 25.1447,E2 474.9654} C_DIS
LIN {X 99.5522,Y -44.0103,Z 111,A -27.496,B 24.9422,C -1.7558,E1 25.1468,E2 473.1838} C_DIS
LIN {X 100.7964,Y -41.0769,Z 111,A -25.5404,B 24.941,C -1.7735,E1 25.1489,E2 471.1973} C_DIS
LIN {X 101.9761,Y -38.0575,Z 111,A -24.3563,B 24.9422,C -1.7554,E1 25.15,E2 470.0624} C_DIS
LIN {X 103.5614,Y -33.5003,Z 111,A -21.7695,B 24.9416,C -1.7655,E1 25.1524,E2 467.4665} C_DIS
LIN {X 104.5197,Y -30.3846,Z 111,A -19.7275,B 24.9402,C -1.7855,E1 25.154,E2 465.389} C_DIS
LIN {X 105.8104,Y -25.524,Z 111,A -17.2596,B 24.9402,C -1.7859,E1 25.1557,E2 462.9343} C_DIS
LIN {X 106.6564,Y -21.7181,Z 111,A -14.2133,B 24.9367,C -1.8374,E1 25.1575,E2 459.7844} C_DIS
LIN {X 107.729,Y -15.548,Z 111,A -11.9826,B 24.9393,C -1.7999,E1 25.1584,E2 457.6552} C_DIS
LIN {X 108.2151,Y -11.6982,Z 111,A -10.0765,B 24.9393,C -1.8004,E1 25.159,E2 455.7591} C_DIS
LIN {X 108.4928,Y -8.7496,Z 111,A -8.4264,B 24.9386,C -1.8096,E1 25.1594,E2 454.0972} C_DIS
LIN {X 108.7396,Y -4.7897,Z 111,A -6.379,B 24.9383,C -1.8145,E1 25.1597,E2 452.0503} C_DIS
LIN {X 108.8406,Y -1.0882,Z 111,A -4.4743,B 24.938,C -1.8189,E1 25.1597,E2 450.1467} C_DIS
LIN {X 108.8216,Y 2.2696,Z 111,A -2.6441,B 24.9374,C -1.8274,E1 25.1597,E2 448.3073} C_DIS
LIN {X 108.678,Y 6.0261,Z 111,A -0.7896,B 24.9374,C -1.8283,E1 25.1595,E2 446.4618} C_DIS
LIN {X 108.4427,Y 9.3706,Z 111,A 1.0773,B 24.9366,C -1.8384,E1 25.1591,E2 444.582} C_DIS
LIN {X 108.093,Y 12.7725,Z 111,A 2.8382,B 24.9364,C -1.8425,E1 25.1585,E2 442.822} C_DIS
LIN {X 107.3579,Y 17.9305,Z 111,A 5.3003,B 24.9366,C -1.8387,E1 25.1575,E2 440.3832} C_DIS
LIN {X 106.1082,Y 24.2557,Z 111,A 8.8283,B 24.9355,C -1.8552,E1 25.1556,E2 436.8369} C_DIS
LIN {X 104.5968,Y 30.1156,Z 111,A 12.5194,B 24.9332,C -1.8875,E1 25.1528,E2 433.0909} C_DIS
LIN {X 103.5848,Y 33.428,Z 111,A 13.8849,B 24.9343,C -1.8726,E1 25.1517,E2 431.7682} C_DIS
LIN {X 102.5326,Y 36.5318,Z 111,A 15.6573,B 24.9338,C -1.8799,E1 25.1501,E2 429.9887} C_DIS
LIN {X 101.3762,Y 39.6247,Z 111,A 17.211,B 24.934,C -1.8769,E1 25.1485,E2 428.4507} C_DIS
LIN {X 100.2808,Y 42.3202,Z 111,A 18.8103,B 24.9334,C -1.8843,E1 25.1468,E2 426.8426} C_DIS
LIN {X 99.005,Y 45.2278,Z 111,A 21.2375,B 24.9307,C -1.9226,E1 25.1439,E2 424.3382} C_DIS
LIN {X 96.9849,Y 49.4082,Z 111,A 22.9524,B 24.9325,C -1.8972,E1 25.1419,E2 422.6926} C_DIS
LIN {X 95.8067,Y 51.6564,Z 111,A 24.9166,B 24.9303,C -1.9286,E1 25.1392,E2 420.6645} C_DIS
LIN {X 93.6611,Y 55.4512,Z 111,A 26.5523,B 24.9319,C -1.9057,E1 25.1369,E2 419.0913} C_DIS
LIN {X 91.7328,Y 58.5866,Z 111,A 28.5306,B 24.9314,C -1.9125,E1 25.134,E2 417.1068} C_DIS
LIN {X 88.76,Y 62.9996,Z 111,A 31.4281,B 24.9306,C -1.9239,E1 25.1294,E2 414.1967} C_DIS
LIN {X 86.2787,Y 66.3569,Z 111,A 33.4015,B 24.9309,C -1.9195,E1 25.1261,E2 412.2429} C_DIS
LIN {X 84.078,Y 69.1263,Z 111,A 35.3296,B 24.9304,C -1.9269,E1 25.1227,E2 410.3066} C_DIS
LIN {X 81.9019,Y 71.689,Z 111,A 37.052,B 24.9302,C -1.9289,E1 25.1196,E2 408.5871} C_DIS
LIN {X 79.3649,Y 74.4879,Z 111,A 39.0654,B 24.9298,C -1.9345,E1 25.1158,E2 406.5694} C_DIS
LIN {X 76.7691,Y 77.1615,Z 111,A 41.0277,B 24.9295,C -1.9387,E1 25.1119,E2 404.6055} C_DIS
LIN {X 74.3517,Y 79.4931,Z 111,A 42.835,B 24.9291,C -1.9441,E1 25.1082,E2 402.7928} C_DIS
LIN {X 71.7358,Y 81.8611,Z 111,A 44.6446,B 24.9291,C -1.9458,E1 25.1045,E2 400.9866} C_DIS
LIN {X 69.8549,Y 83.4726,Z 111,A 46.598,B 24.9268,C -1.9764,E1 25.1001,E2 398.9684} C_DIS
LIN {X 66.3078,Y 86.3165,Z 111,A 48.3257,B 24.9286,C -1.952,E1 25.0965,E2 397.3046} C_DIS
LIN {X 63.3645,Y 88.4997,Z 111,A 50.2386,B 24.9284,C -1.9547,E1 25.0921,E2 395.3922} C_DIS
LIN {X 60.2993,Y 90.617,Z 111,A 52.0826,B 24.9284,C -1.9529,E1 25.0879,E2 393.5586} C_DIS
Enddeposition()
END
